	//Delete counters
	IF "DB_ProductionCountersEdit".DeleteCounters > 0 AND "DB_ProductionCountersEdit".DeleteCounters < 4 THEN
	    IF "DB_ProductionCountersEdit".ProgramNumber > 0 AND "DB_ProductionCountersEdit".ProgramNumber <= "NumberOfProductionPrograms" THEN
	        #shiftToDelete := "DB_ProductionCountersEdit".DeleteCounters;
	        "DB_ProductionCountersList".Program["DB_ProductionCountersEdit".ProgramNumber].Product[1].Shift[#shiftToDelete].Ok := 0;
	        "DB_ProductionCountersList".Program["DB_ProductionCountersEdit".ProgramNumber].Product[1].Shift[#shiftToDelete].Nok := 0;
	        "DB_ProductionCountersEdit".ProductCounters := "DB_ProductionCountersList".Program["DB_ProductionCountersEdit".ProgramNumber];
	        FOR #i := 1 TO 50 DO
	            "PartErrorsCounter".CountersRef["DB_ProductionCountersEdit".ProgramNumber].Counters[#shiftToDelete, #i] := 0;
	        END_FOR;
	    END_IF;
	    "DB_ProductionCountersEdit".DeleteCounters := 0;
	END_IF;
	        
	    
	//Auto reset shift counters
	IF "DB_DateTimeAndShifts_Instance".ShiftStatus.Shift1Started THEN
	    FOR #i := 1 TO "NumberOfProductionPrograms" DO
	        "DB_ProductionCountersList".Program[#i].Product[1].Shift[1].Ok := 0;
	        "DB_ProductionCountersList".Program[#i].Product[1].Shift[1].Nok := 0;
	    END_FOR;
	END_IF;
	IF "DB_DateTimeAndShifts_Instance".ShiftStatus.Shift2Started THEN
	    FOR #i := 1 TO "NumberOfProductionPrograms" DO
	        "DB_ProductionCountersList".Program[#i].Product[1].Shift[2].Ok := 0;
	        "DB_ProductionCountersList".Program[#i].Product[1].Shift[2].Nok := 0;
	    END_FOR;
	END_IF;
	IF "DB_DateTimeAndShifts_Instance".ShiftStatus.Shift3Started THEN
	    FOR #i := 1 TO "NumberOfProductionPrograms" DO
	        "DB_ProductionCountersList".Program[#i].Product[1].Shift[3].Ok := 0;
	        "DB_ProductionCountersList".Program[#i].Product[1].Shift[3].Nok := 0;
	    END_FOR;
	END_IF;
	
END_FUNCTION_BLOCK

FUNCTION "PartErrorsCountersMain" : Void
{ S7_Optimized_Access := 'TRUE' }
VERSION : 0.1
   VAR_TEMP 
      i : Int;
   END_VAR


BEGIN
	IF "DB_ProductionCountersEdit".ProgramNumber > 0 AND "DB_ProductionCountersEdit".ProgramNumber <= "NumberOfProductionPrograms" THEN
	    "PartErrorsCounter".CountersHMI := "PartErrorsCounter".CountersRef["DB_ProductionCountersEdit".ProgramNumber];
	END_IF;
	
	
	
	
	
	
	
END_FUNCTION

FUNCTION_BLOCK "FB_Devices"   // FB5100, LAD
{ S7_Optimized_Access := 'TRUE' }
VERSION : 0.1
// stored: AutoNumber false, IsIECCheckEnabled false, IsRetainMemResEnabled false, MemoryReserve 100, SetENOAutomatically false, UDAEnableTagReadback false
   VAR
      ServiceDoors_Instance_1 { S7_SetPoint := 'True'} : "serviceDoor";
      ServiceDoors_Instance_2 { S7_SetPoint := 'True'} : "serviceDoor";
      R_TRIG_Instance { S7_SetPoint := 'True'} : R_TRIG;
      HydraulicActive { S7_SetPoint := 'True'} : Bool;
      HydraulicActiveOffMem : Bool;
      HydraulicOnMem : Bool;
      IEC_Timer_0_Instance { S7_SetPoint := 'True'} : TON_TIME;
      IEC_Timer_0_Instance_1 { S7_SetPoint := 'True'} : TON_TIME;
      FB_TurnTable_Instance { S7_SetPoint := 'True'} : "FB_TurnTable";
      F_TRIG_Instance { S7_SetPoint := 'True'} : F_TRIG;
      edges { S7_SetPoint := 'True'} : Array[1..6] of Bool;
      ManualCommandOld : Int;
      R_TRIG_Instance_1 { S7_SetPoint := 'True'} : R_TRIG;
      R_TRIG_Instance_2 { S7_SetPoint := 'True'} : R_TRIG;
      R_TRIG_Instance_3 { S7_SetPoint := 'True'} : R_TRIG;
      R_TRIG_Instance_4 { S7_SetPoint := 'True'} : R_TRIG;
      R_TRIG_Instance_6 { S7_SetPoint := 'True'} : R_TRIG;
      R_TRIG_Instance_7 { S7_SetPoint := 'True'} : R_TRIG;
      R_TRIG_Instance_8 { S7_SetPoint := 'True'} : R_TRIG;
      R_TRIG_Instance_5 { S7_SetPoint := 'True'} : R_TRIG;
      edgesFitting : Array[1..4] of Bool;
      R_TRIG_V240Wp { S7_SetPoint := 'True'} : R_TRIG;
      R_TRIG_V240Bp { S7_SetPoint := 'True'} : R_TRIG;
      ReaderKeyence_Instance { S7_SetPoint := 'True'} : "ReaderKeyence";
      IEC_Timer_0_Instance_2 { S7_SetPoint := 'True'} : TON_TIME;
      FriedrichUnit1_Instance { S7_SetPoint := 'True'} : "FriedrichUnit";
      FriedrichUnit2_Instance { S7_SetPoint := 'True'} : "FriedrichUnit";
      Trig1 { S7_SetPoint := 'True'} : R_TRIG;
      Trig2 { S7_SetPoint := 'True'} : R_TRIG;
      Trig3 { S7_SetPoint := 'True'} : R_TRIG;
      Trig4 { S7_SetPoint := 'True'} : R_TRIG;
      Camera_CAM1 { S7_SetPoint := 'True'} : "Camera";
      Camera_CAM2 { S7_SetPoint := 'True'} : "Camera";
      Camera_CAM3 { S7_SetPoint := 'True'} : "Camera";
      Camera_CAM4 { S7_SetPoint := 'True'} : "Camera";
      RivetingCycleLeft_Instance { S7_SetPoint := 'True'} : "RivetingCycle";
      RivetingCycleRight_Instance { S7_SetPoint := 'True'} : "RivetingCycle";
   END_VAR
   VAR_TEMP
      posTemp : "UDT_PositionData";
      i : Int;
   END_VAR
   VAR_TEMP   // added for the SCL form of the ladder/FBD networks
      _w1 : Bool;
      _w2 : Bool;
      _w3 : Bool;
   END_VAR
BEGIN

REGION Network 1: Diagnostic fieldbus devices
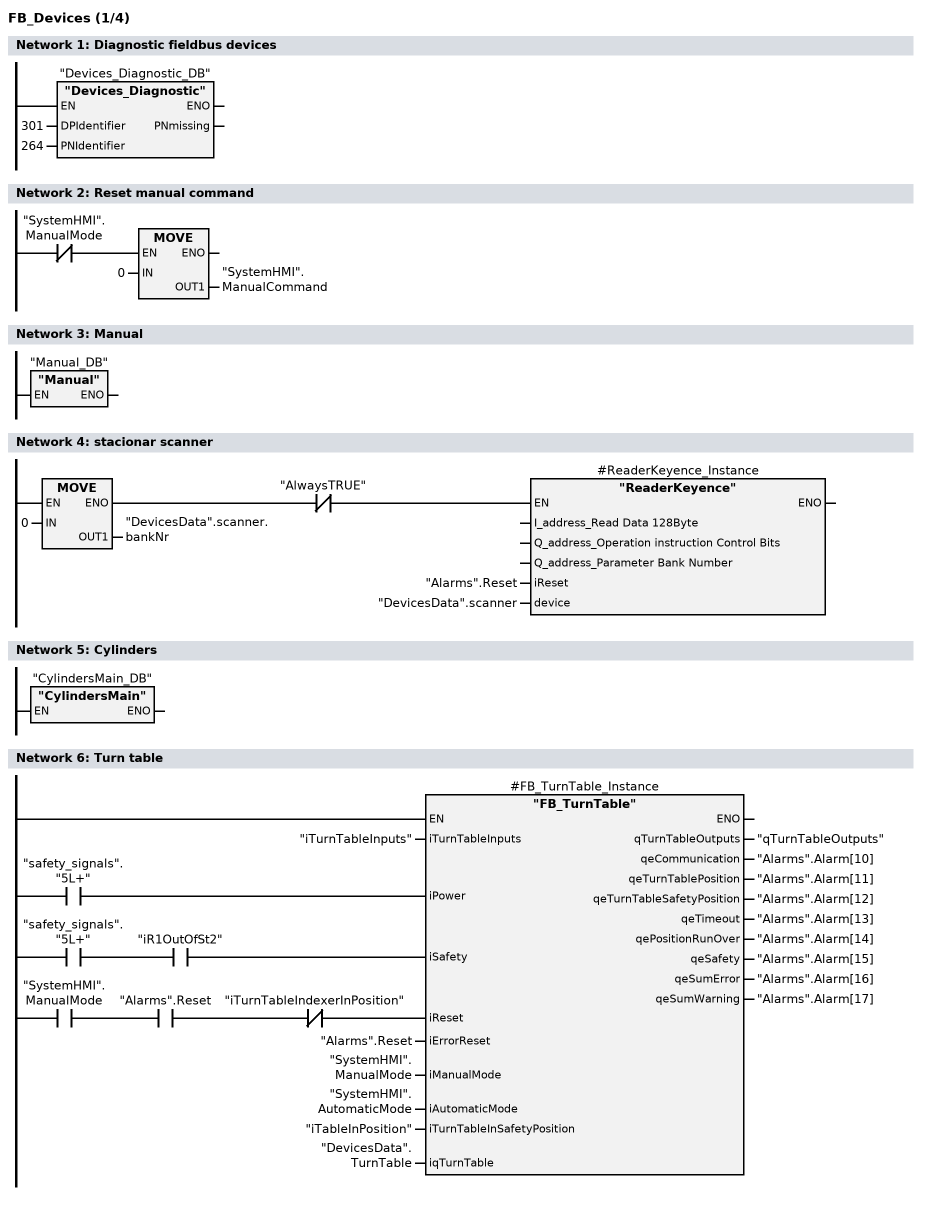
   RUNG wire#powerrail
      "Devices_Diagnostic_DB"(DPIdentifier := 301, PNIdentifier := 264, PNmissing =>)
   END_RUNG
   // the same network as SCL:
   "Devices_Diagnostic_DB"(DPIdentifier := 301, PNIdentifier := 264);   // "Devices_Diagnostic"
END_REGION

REGION Network 2: Reset manual command
   RUNG wire#powerrail
      I_Contact( "SystemHMI".ManualMode )
      Move(in := 0, out1 => "SystemHMI".ManualCommand)
   END_RUNG
   // the same network as SCL:
   IF NOT "SystemHMI".ManualMode THEN "SystemHMI".ManualCommand := 0; END_IF;
END_REGION

REGION Network 3: Manual
   RUNG wire#powerrail
      "Manual_DB"()
   END_RUNG
   // the same network as SCL:
   "Manual_DB"();   // "Manual"
END_REGION

REGION Network 4: stacionar scanner
   RUNG wire#powerrail
      Move(in := 0, out1 => "DevicesData".scanner.bankNr)
      I_Contact( "AlwaysTRUE" )
      #ReaderKeyence_Instance("I_address_Read Data 128Byte" :=, "Q_address_Operation instruction Control Bits" :=, "Q_address_Parameter Bank Number" :=, iReset := "Alarms".Reset, device := "DevicesData".scanner)
   END_RUNG
   // the same network as SCL:
   "DevicesData".scanner.bankNr := 0;
   IF NOT "AlwaysTRUE" THEN
       #ReaderKeyence_Instance(iReset := "Alarms".Reset, device := "DevicesData".scanner);   // "ReaderKeyence"
   END_IF;
END_REGION

REGION Network 5: Cylinders
   RUNG wire#powerrail
      "CylindersMain_DB"()
   END_RUNG
   // the same network as SCL:
   "CylindersMain_DB"();   // "CylindersMain"
END_REGION

REGION Network 6: Turn table
   RUNG wire#powerrail
      #FB_TurnTable_Instance(iPower := wire#w1, iSafety := wire#w2, iReset := wire#w3, iTurnTableInputs := "iTurnTableInputs", iErrorReset := "Alarms".Reset, iManualMode := "SystemHMI".ManualMode, iAutomaticMode := "SystemHMI".AutomaticMode, iTurnTableInSafetyPosition := "iTableInPosition", iqTurnTable := "DevicesData".TurnTable, qTurnTableOutputs => "qTurnTableOutputs", qeCommunication => "Alarms".Alarm[10], qeTurnTablePosition => "Alarms".Alarm[11], qeTurnTableSafetyPosition => "Alarms".Alarm[12], qeTimeout => "Alarms".Alarm[13], qePositionRunOver => "Alarms".Alarm[14], qeSafety => "Alarms".Alarm[15], qeSumError => "Alarms".Alarm[16], qeSumWarning => "Alarms".Alarm[17])
   END_RUNG
   RUNG wire#powerrail
      Contact( "safety_signals"."5L+" )
   END_RUNG wire#w1
   RUNG wire#powerrail
      Contact( "safety_signals"."5L+" )
      Contact( "iR1OutOfSt2" )
   END_RUNG wire#w2
   RUNG wire#powerrail
      Contact( "SystemHMI".ManualMode )
      Contact( "Alarms".Reset )
      I_Contact( "iTurnTableIndexerInPosition" )
   END_RUNG wire#w3
   // the same network as SCL:
   #FB_TurnTable_Instance(iTurnTableInputs := "iTurnTableInputs",   // "FB_TurnTable"
                          iPower := "safety_signals"."5L+",
                          iSafety := "safety_signals"."5L+" AND "iR1OutOfSt2",
                          iReset := "SystemHMI".ManualMode AND "Alarms".Reset AND NOT "iTurnTableIndexerInPosition",
                          iErrorReset := "Alarms".Reset,
                          iManualMode := "SystemHMI".ManualMode,
                          iAutomaticMode := "SystemHMI".AutomaticMode,
                          iTurnTableInSafetyPosition := "iTableInPosition",
                          iqTurnTable := "DevicesData".TurnTable,
                          qTurnTableOutputs => "qTurnTableOutputs",
                          qeCommunication => "Alarms".Alarm[10],
                          qeTurnTablePosition => "Alarms".Alarm[11],
                          qeTurnTableSafetyPosition => "Alarms".Alarm[12],
                          qeTimeout => "Alarms".Alarm[13],
                          qePositionRunOver => "Alarms".Alarm[14],
                          qeSafety => "Alarms".Alarm[15],
                          qeSumError => "Alarms".Alarm[16],
                          qeSumWarning => "Alarms".Alarm[17]);
END_REGION

REGION Network 7: Handle table positions
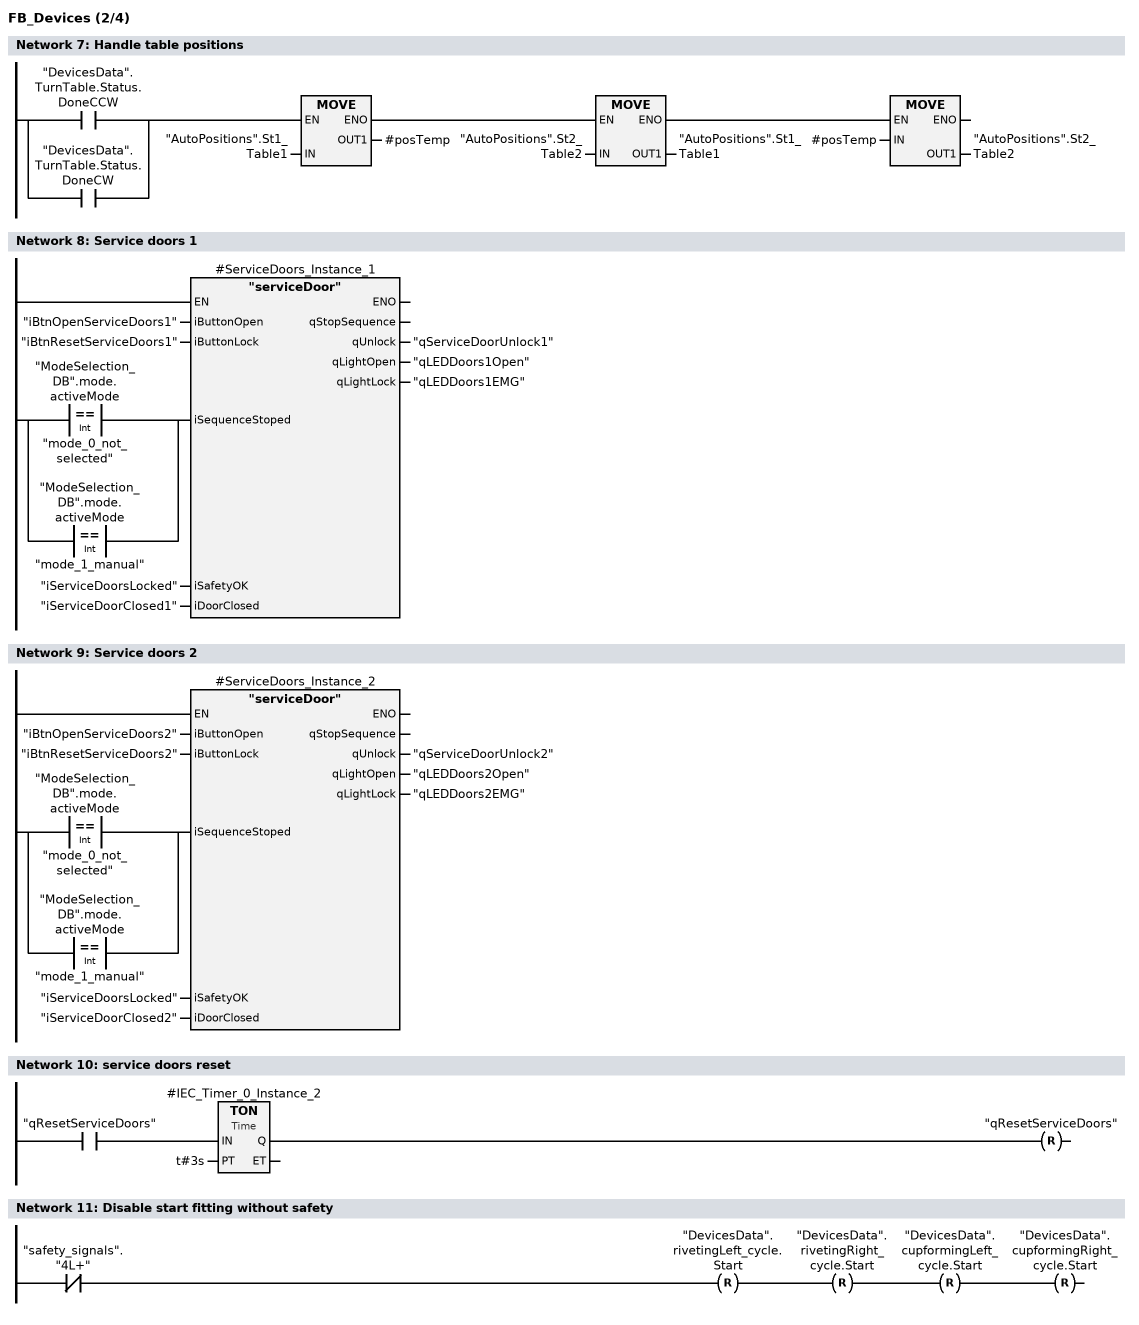
   RUNG wire#powerrail
      Contact( "DevicesData".TurnTable.Status.DoneCCW )
      wire#w1
      Move(in := "AutoPositions".St1_Table1, out1 => #posTemp)
      Move(in := "AutoPositions".St2_Table2, out1 => "AutoPositions".St1_Table1)
      Move(in := #posTemp, out1 => "AutoPositions".St2_Table2)
   END_RUNG
   RUNG wire#powerrail
      Contact( "DevicesData".TurnTable.Status.DoneCW )
   END_RUNG wire#w1
   // the same network as SCL:
   IF "DevicesData".TurnTable.Status.DoneCCW OR "DevicesData".TurnTable.Status.DoneCW THEN
       #posTemp := "AutoPositions".St1_Table1;
       "AutoPositions".St1_Table1 := "AutoPositions".St2_Table2;
       "AutoPositions".St2_Table2 := #posTemp;
   END_IF;
END_REGION

REGION Network 8: Service doors 1
   RUNG wire#powerrail
      #ServiceDoors_Instance_1(iSequenceStoped := wire#w1, iButtonOpen := "iBtnOpenServiceDoors1", iButtonLock := "iBtnResetServiceDoors1", iSafetyOK := "iServiceDoorsLocked", iDoorClosed := "iServiceDoorClosed1", qStopSequence =>, qUnlock => "qServiceDoorUnlock1", qLightOpen => "qLEDDoors1Open", qLightLock => "qLEDDoors1EMG")
   END_RUNG
   RUNG wire#powerrail
      { S7_Templates := "SrcType := Int" } EQ_Contact(in1 := "ModeSelection_DB".mode.activeMode, in2 := "mode_0_not_selected")
   END_RUNG wire#w1
   RUNG wire#powerrail
      { S7_Templates := "SrcType := Int" } EQ_Contact(in1 := "ModeSelection_DB".mode.activeMode, in2 := "mode_1_manual")
   END_RUNG wire#w1
   // the same network as SCL:
   #ServiceDoors_Instance_1(iButtonOpen := "iBtnOpenServiceDoors1",   // "serviceDoor"
                           iButtonLock := "iBtnResetServiceDoors1",
                           iSequenceStoped := ("ModeSelection_DB".mode.activeMode = "mode_0_not_selected") OR ("ModeSelection_DB".mode.activeMode = "mode_1_manual"),
                           iSafetyOK := "iServiceDoorsLocked",
                           iDoorClosed := "iServiceDoorClosed1",
                           qUnlock => "qServiceDoorUnlock1",
                           qLightOpen => "qLEDDoors1Open",
                           qLightLock => "qLEDDoors1EMG");
END_REGION

REGION Network 9: Service doors 2
   RUNG wire#powerrail
      #ServiceDoors_Instance_2(iSequenceStoped := wire#w1, iButtonOpen := "iBtnOpenServiceDoors2", iButtonLock := "iBtnResetServiceDoors2", iSafetyOK := "iServiceDoorsLocked", iDoorClosed := "iServiceDoorClosed2", qStopSequence =>, qUnlock => "qServiceDoorUnlock2", qLightOpen => "qLEDDoors2Open", qLightLock => "qLEDDoors2EMG")
   END_RUNG
   RUNG wire#powerrail
      { S7_Templates := "SrcType := Int" } EQ_Contact(in1 := "ModeSelection_DB".mode.activeMode, in2 := "mode_0_not_selected")
   END_RUNG wire#w1
   RUNG wire#powerrail
      { S7_Templates := "SrcType := Int" } EQ_Contact(in1 := "ModeSelection_DB".mode.activeMode, in2 := "mode_1_manual")
   END_RUNG wire#w1
   // the same network as SCL:
   #ServiceDoors_Instance_2(iButtonOpen := "iBtnOpenServiceDoors2",   // "serviceDoor"
                           iButtonLock := "iBtnResetServiceDoors2",
                           iSequenceStoped := ("ModeSelection_DB".mode.activeMode = "mode_0_not_selected") OR ("ModeSelection_DB".mode.activeMode = "mode_1_manual"),
                           iSafetyOK := "iServiceDoorsLocked",
                           iDoorClosed := "iServiceDoorClosed2",
                           qUnlock => "qServiceDoorUnlock2",
                           qLightOpen => "qLEDDoors2Open",
                           qLightLock => "qLEDDoors2EMG");
END_REGION

REGION Network 10: service doors reset
   RUNG wire#powerrail
      Contact( "qResetServiceDoors" )
      { S7_Templates := "time_type := Time" } #IEC_Timer_0_Instance_2.TON(pt := t#3s, et =>)
      R_Coil( "qResetServiceDoors" )
   END_RUNG
   // the same network as SCL:
   #IEC_Timer_0_Instance_2(IN := "qResetServiceDoors", PT := t#3s);   // TON
   IF #IEC_Timer_0_Instance_2.Q THEN "qResetServiceDoors" := FALSE; END_IF;
END_REGION

REGION Network 11: Disable start fitting without safety
   RUNG wire#powerrail
      I_Contact( "safety_signals"."4L+" )
      R_Coil( "DevicesData".rivetingLeft_cycle.Start )
      R_Coil( "DevicesData".rivetingRight_cycle.Start )
      R_Coil( "DevicesData".cupformingLeft_cycle.Start )
      R_Coil( "DevicesData".cupformingRight_cycle.Start )
   END_RUNG
   // the same network as SCL:
   IF NOT "safety_signals"."4L+" THEN
       "DevicesData".rivetingLeft_cycle.Start := FALSE;
       "DevicesData".rivetingRight_cycle.Start := FALSE;
       "DevicesData".cupformingLeft_cycle.Start := FALSE;
       "DevicesData".cupformingRight_cycle.Start := FALSE;
   END_IF;
END_REGION

REGION Network 12: Fittings - Cyle times measurement
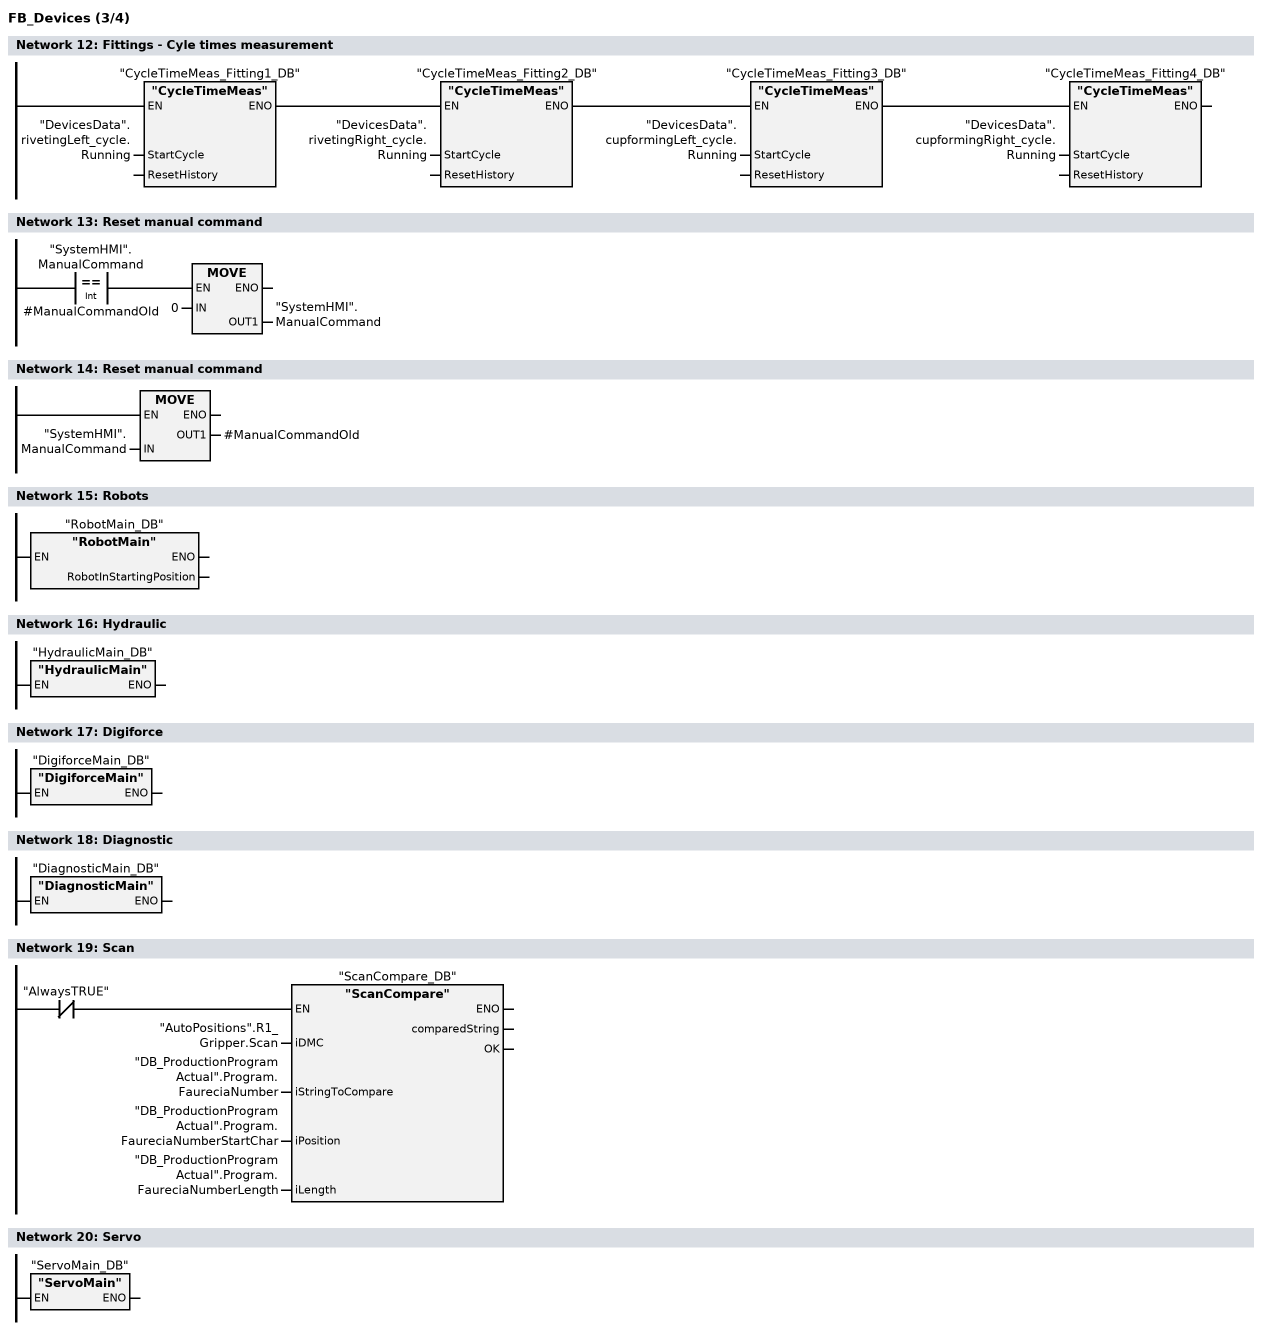
   RUNG wire#powerrail
      "CycleTimeMeas_Fitting1_DB"(StartCycle := "DevicesData".rivetingLeft_cycle.Running, ResetHistory :=)
      "CycleTimeMeas_Fitting2_DB"(StartCycle := "DevicesData".rivetingRight_cycle.Running, ResetHistory :=)
      "CycleTimeMeas_Fitting3_DB"(StartCycle := "DevicesData".cupformingLeft_cycle.Running, ResetHistory :=)
      "CycleTimeMeas_Fitting4_DB"(StartCycle := "DevicesData".cupformingRight_cycle.Running, ResetHistory :=)
   END_RUNG
   // the same network as SCL:
   "CycleTimeMeas_Fitting1_DB"(StartCycle := "DevicesData".rivetingLeft_cycle.Running, ENO => #_w1);   // "CycleTimeMeas"
   "CycleTimeMeas_Fitting2_DB"(EN := #_w1, StartCycle := "DevicesData".rivetingRight_cycle.Running, ENO => #_w2);   // "CycleTimeMeas"
   "CycleTimeMeas_Fitting3_DB"(EN := #_w2,   // "CycleTimeMeas"
                           StartCycle := "DevicesData".cupformingLeft_cycle.Running,
                           ENO => #_w3);
   IF #_w3 THEN
       "CycleTimeMeas_Fitting4_DB"(StartCycle := "DevicesData".cupformingRight_cycle.Running);   // "CycleTimeMeas"
   END_IF;
END_REGION

REGION Network 13: Reset manual command
   RUNG wire#powerrail
      { S7_Templates := "SrcType := Int" } EQ_Contact(in1 := "SystemHMI".ManualCommand, in2 := #ManualCommandOld)
      Move(in := 0, out1 => "SystemHMI".ManualCommand)
   END_RUNG
   // the same network as SCL:
   IF "SystemHMI".ManualCommand = #ManualCommandOld THEN "SystemHMI".ManualCommand := 0; END_IF;
END_REGION

REGION Network 14: Reset manual command
   RUNG wire#powerrail
      Move(in := "SystemHMI".ManualCommand, out1 => #ManualCommandOld)
   END_RUNG
   // the same network as SCL:
   #ManualCommandOld := "SystemHMI".ManualCommand;
END_REGION

REGION Network 15: Robots
   RUNG wire#powerrail
      "RobotMain_DB"(RobotInStartingPosition =>)
   END_RUNG
   // the same network as SCL:
   "RobotMain_DB"();   // "RobotMain"
END_REGION

REGION Network 16: Hydraulic
   RUNG wire#powerrail
      "HydraulicMain_DB"()
   END_RUNG
   // the same network as SCL:
   "HydraulicMain_DB"();   // "HydraulicMain"
END_REGION

REGION Network 17: Digiforce
   RUNG wire#powerrail
      "DigiforceMain_DB"()
   END_RUNG
   // the same network as SCL:
   "DigiforceMain_DB"();   // "DigiforceMain"
END_REGION

REGION Network 18: Diagnostic
   RUNG wire#powerrail
      "DiagnosticMain_DB"()
   END_RUNG
   // the same network as SCL:
   "DiagnosticMain_DB"();   // "DiagnosticMain"
END_REGION

REGION Network 19: Scan
   RUNG wire#powerrail
      I_Contact( "AlwaysTRUE" )
      "ScanCompare_DB"(iDMC := "AutoPositions".R1_Gripper.Scan, iStringToCompare := "DB_ProductionProgramActual".Program.FaureciaNumber, iPosition := "DB_ProductionProgramActual".Program.FaureciaNumberStartChar, iLength := "DB_ProductionProgramActual".Program.FaureciaNumberLength, comparedString =>, OK =>)
   END_RUNG
   // the same network as SCL:
   IF NOT "AlwaysTRUE" THEN
       "ScanCompare_DB"(iDMC := "AutoPositions".R1_Gripper.Scan,   // "ScanCompare"
                        iStringToCompare := "DB_ProductionProgramActual".Program.FaureciaNumber,
                        iPosition := "DB_ProductionProgramActual".Program.FaureciaNumberStartChar,
                        iLength := "DB_ProductionProgramActual".Program.FaureciaNumberLength);
   END_IF;
END_REGION

REGION Network 20: Servo
   RUNG wire#powerrail
      "ServoMain_DB"()
   END_RUNG
   // the same network as SCL:
   "ServoMain_DB"();   // "ServoMain"
END_REGION

REGION Network 21 (SCL): Friedrich1 R
   IF "HMIData".ManualCommand = 611 THEN
       "DevicesData".Friedrich1.Start := true;
   END_IF;

   #FriedrichUnit1_Instance(safetyOK := "safety_signals"."4L+",
                            iReady := "iRivetingReady1",
                            iZ1OK := "iRivetingZ1ok1",
                            iH1OK := "iRivetingH1ok1",
                            iH2OK := "iRivetingH2ok1",
                            iTimeOK := "iRivetingTimeOk1",
                            iNoAlarm := "iRivetingNoError1",
                            FriedrichNumber := 1,
                            Port := 39000,
                            IP1 := 192,
                            IP2 := 168,
                            IP3 := 16,
                            IP4 := 43,
                            ID := 2,
                            qStart => "qRiveting1Start",
                            qPrgbit4 => "qRiveting1Bit4",
                            qPrgbit3 => "qRiveting1Bit3",
                            qPrgbit2 => "qRiveting1Bit2",
                            qPrgbit1 => "qRiveting1Bit1",
                            qPrgbit0 => "qRiveting1Bit0",
                            RivetData := "DevicesData".Friedrich1);
   "qFriedrich1_setup_mode" := "DB_MainData".MachineMode <> 2 AND "DB_MainData".MachineMode <> 3;

   #Trig1(CLK:="DevicesData".Friedrich1.OK);
   #Trig2(CLK:="DevicesData".Friedrich1.NOK);
   "RivetingHistoryRight_DB"(iNewCycle := #Trig1.Q OR #Trig2.Q,
                             iData := "DevicesData".Friedrich1);

   #RivetingCycleRight_Instance(parameters := "DB_ProductionProgramActual".Program.Riveting_program_right,
                                basicPosition := "DevicesData".Friedrich1.Ready AND "DevicesData".Cylinders[MM340_RivetingUnitRight].InBp AND "DevicesData".Cylinders[MM344_RivetingSupportRight].InBp,
                                twoRivets := "DB_ProductionProgramActual".Program.Total_number_of_rivets_4,
                                MeasuredData1=>"AutoInfo".PartMeasuredData.RightRiveting1,
                                MeasuredData2=>"AutoInfo".PartMeasuredData.RightRiveting2,
                                riveter := "DevicesData".Friedrich1,
                                data := "DevicesData".rivetingRight_cycle,
                                cylinderSupport := "DevicesData".Cylinders[MM344_RivetingSupportRight],
                                cylinderShift := "DevicesData".Cylinders[MM340_RivetingUnitRight]);
END_REGION

REGION Network 22 (SCL): Friedrich2 L
   IF "HMIData".ManualCommand = 612 THEN
       "DevicesData".Friedrich2.Start := true;
   END_IF;
   #FriedrichUnit2_Instance(safetyOK := "safety_signals"."4L+",
                            iReady := "iRivetingReady2",
                            iZ1OK := "iRivetingZ1ok2",
                            iH1OK := "iRivetingH1ok2",
                            iH2OK := "iRivetingH2ok2",
                            iTimeOK := "iRivetingTimeOk2",
                            iNoAlarm := "iRivetingNoError2",
                            FriedrichNumber := 2,
                            Port := 39000,
                            IP1 := 192,
                            IP2 := 168,
                            IP3 := 16,
                            IP4 := 44,
                            ID := 3,
                            qStart => "qRiveting2Start",
                            qPrgbit4 => "qRiveting2Bit4",
                            qPrgbit3 => "qRiveting2Bit3",
                            qPrgbit2 => "qRiveting2Bit2",
                            qPrgbit1 => "qRiveting2Bit1",
                            qPrgbit0 => "qRiveting2Bit0",
                            RivetData := "DevicesData".Friedrich2);
   "qFriedrich2_setup_mode" := "DB_MainData".MachineMode <> 2 AND "DB_MainData".MachineMode <> 3;

   #Trig3(CLK:="DevicesData".Friedrich2.OK);
   #Trig4(CLK:="DevicesData".Friedrich2.NOK);
   "RivetingHistoryLeft_DB"(iNewCycle := #Trig3.Q OR #Trig4.Q,
                            iData := "DevicesData".Friedrich2);

   #RivetingCycleLeft_Instance(parameters := "DB_ProductionProgramActual".Program.Riveting_program_left,
                               basicPosition := "DevicesData".Friedrich2.Ready AND "DevicesData".Cylinders[MM342_RivetingUnitLeft].InBp AND "DevicesData".Cylinders[MM346_RivetingSupportLeft].InBp,
                               twoRivets := "DB_ProductionProgramActual".Program.Total_number_of_rivets_4,
                               MeasuredData1=>"AutoInfo".PartMeasuredData.LeftRiveting1,
                               MeasuredData2=>"AutoInfo".PartMeasuredData.LeftRiveting2,
                               riveter := "DevicesData".Friedrich2,
                               data := "DevicesData".rivetingLeft_cycle,
                               cylinderSupport := "DevicesData".Cylinders[MM346_RivetingSupportLeft],
                               cylinderShift := "DevicesData".Cylinders[MM342_RivetingUnitLeft]);

   REGION cycles handshake
       IF "SystemHMI".AutomaticMode THEN
           IF "DevicesData".cupformingLeft_cycle.Done AND "DevicesData".cupformingRight_cycle.Done THEN
               "DevicesData".rivetingLeft_cycle.ContinueFitting := TRUE;
               "DevicesData".rivetingRight_cycle.ContinueFitting := TRUE;
           END_IF;
       END_IF;
       "DevicesData".rivetingLeft_cycle.ContinueFitting := TRUE;
       "DevicesData".rivetingRight_cycle.ContinueFitting := TRUE;

       IF "SystemHMI".ManualMode THEN
           "DevicesData".rivetingLeft_cycle.ContinueFitting := true;
           "DevicesData".rivetingRight_cycle.ContinueFitting := true;
       END_IF;
   END_REGION
END_REGION

REGION Network 23
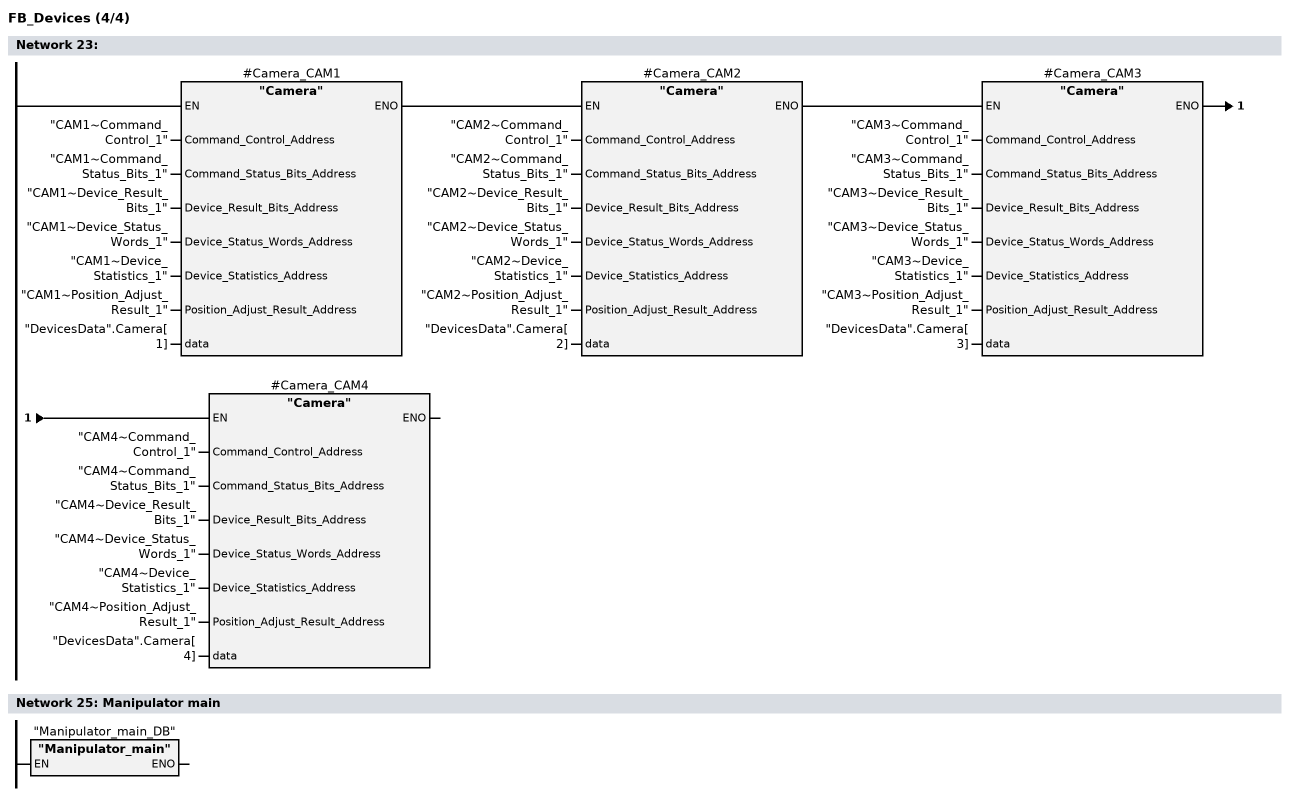
   RUNG wire#powerrail
      #Camera_CAM1(Command_Control_Address := "CAM1~Command_Control_1", Command_Status_Bits_Address := "CAM1~Command_Status_Bits_1", Device_Result_Bits_Address := "CAM1~Device_Result_Bits_1", Device_Status_Words_Address := "CAM1~Device_Status_Words_1", Device_Statistics_Address := "CAM1~Device_Statistics_1", Position_Adjust_Result_Address := "CAM1~Position_Adjust_Result_1", data := "DevicesData".Camera[1])
      #Camera_CAM2(Command_Control_Address := "CAM2~Command_Control_1", Command_Status_Bits_Address := "CAM2~Command_Status_Bits_1", Device_Result_Bits_Address := "CAM2~Device_Result_Bits_1", Device_Status_Words_Address := "CAM2~Device_Status_Words_1", Device_Statistics_Address := "CAM2~Device_Statistics_1", Position_Adjust_Result_Address := "CAM2~Position_Adjust_Result_1", data := "DevicesData".Camera[2])
      #Camera_CAM3(Command_Control_Address := "CAM3~Command_Control_1", Command_Status_Bits_Address := "CAM3~Command_Status_Bits_1", Device_Result_Bits_Address := "CAM3~Device_Result_Bits_1", Device_Status_Words_Address := "CAM3~Device_Status_Words_1", Device_Statistics_Address := "CAM3~Device_Statistics_1", Position_Adjust_Result_Address := "CAM3~Position_Adjust_Result_1", data := "DevicesData".Camera[3])
      #Camera_CAM4(Command_Control_Address := "CAM4~Command_Control_1", Command_Status_Bits_Address := "CAM4~Command_Status_Bits_1", Device_Result_Bits_Address := "CAM4~Device_Result_Bits_1", Device_Status_Words_Address := "CAM4~Device_Status_Words_1", Device_Statistics_Address := "CAM4~Device_Statistics_1", Position_Adjust_Result_Address := "CAM4~Position_Adjust_Result_1", data := "DevicesData".Camera[4])
   END_RUNG
   // the same network as SCL:
   #Camera_CAM1(Command_Control_Address := "CAM1~Command_Control_1",   // "Camera"
                Command_Status_Bits_Address := "CAM1~Command_Status_Bits_1",
                Device_Result_Bits_Address := "CAM1~Device_Result_Bits_1",
                Device_Status_Words_Address := "CAM1~Device_Status_Words_1",
                Device_Statistics_Address := "CAM1~Device_Statistics_1",
                Position_Adjust_Result_Address := "CAM1~Position_Adjust_Result_1",
                data := "DevicesData".Camera[1],
                ENO => #_w1);
   #Camera_CAM2(EN := #_w1,   // "Camera"
                Command_Control_Address := "CAM2~Command_Control_1",
                Command_Status_Bits_Address := "CAM2~Command_Status_Bits_1",
                Device_Result_Bits_Address := "CAM2~Device_Result_Bits_1",
                Device_Status_Words_Address := "CAM2~Device_Status_Words_1",
                Device_Statistics_Address := "CAM2~Device_Statistics_1",
                Position_Adjust_Result_Address := "CAM2~Position_Adjust_Result_1",
                data := "DevicesData".Camera[2],
                ENO => #_w2);
   #Camera_CAM3(EN := #_w2,   // "Camera"
                Command_Control_Address := "CAM3~Command_Control_1",
                Command_Status_Bits_Address := "CAM3~Command_Status_Bits_1",
                Device_Result_Bits_Address := "CAM3~Device_Result_Bits_1",
                Device_Status_Words_Address := "CAM3~Device_Status_Words_1",
                Device_Statistics_Address := "CAM3~Device_Statistics_1",
                Position_Adjust_Result_Address := "CAM3~Position_Adjust_Result_1",
                data := "DevicesData".Camera[3],
                ENO => #_w3);
   IF #_w3 THEN
       #Camera_CAM4(Command_Control_Address := "CAM4~Command_Control_1",   // "Camera"
                    Command_Status_Bits_Address := "CAM4~Command_Status_Bits_1",
                    Device_Result_Bits_Address := "CAM4~Device_Result_Bits_1",
                    Device_Status_Words_Address := "CAM4~Device_Status_Words_1",
                    Device_Statistics_Address := "CAM4~Device_Statistics_1",
                    Position_Adjust_Result_Address := "CAM4~Position_Adjust_Result_1",
                    data := "DevicesData".Camera[4]);
   END_IF;
END_REGION

REGION Network 24 (SCL)
   "DevicesData".Camera[1].ProgramNumber := USINT_TO_SINT("DB_ProductionProgramActual".Program.Camera_program[1]);
   "DevicesData".Camera[2].ProgramNumber := USINT_TO_SINT("DB_ProductionProgramActual".Program.Camera_program[2]);
   "DevicesData".Camera[3].ProgramNumber := USINT_TO_SINT("DB_ProductionProgramActual".Program.Camera_program[3]);
   "DevicesData".Camera[4].ProgramNumber := USINT_TO_SINT("DB_ProductionProgramActual".Program.Camera_program[4]);
END_REGION

REGION Network 25: Manipulator main
   RUNG wire#powerrail
      "Manipulator_main_DB"()
   END_RUNG
   // the same network as SCL:
   "Manipulator_main_DB"();   // "Manipulator_main"
END_REGION

REGION Network 26: Readers
END_REGION
END_FUNCTION_BLOCK

FUNCTION_BLOCK "Devices_Diagnostic"
{ S7_Optimized_Access := 'TRUE' }
VERSION : 0.1
   VAR_INPUT 
      DPIdentifier : HW_IOSYSTEM;
      PNIdentifier : HW_IOSYSTEM;
   END_VAR

   VAR_OUTPUT 
      PNmissing : Bool;
   END_VAR

   VAR 
      PNConfigured : Array[0..1023] of Bool;
      PNFaulty : Array[0..1023] of Bool;
      PNDisabled : Array[0..1023] of Bool;
      PNExist : Array[0..1023] of Bool;
      DPConfigured : Array[0..1023] of Bool;
      DPFaulty : Array[0..1023] of Bool;
      DPDisabled : Array[0..1023] of Bool;
      DPExist : Array[0..1023] of Bool;
   END_VAR

   VAR_TEMP 
      ret : Int;
   END_VAR


BEGIN
	IF #PNIdentifier > 0 THEN
	    #ret := DeviceStates(LADDR := #PNIdentifier, MODE := 1, STATE := #PNConfigured);
	    #ret := DeviceStates(LADDR := #PNIdentifier, MODE := 2, STATE := #PNFaulty);
	    #ret := DeviceStates(LADDR := #PNIdentifier, MODE := 3, STATE := #PNDisabled);
	    #ret := DeviceStates(LADDR := #PNIdentifier, MODE := 4, STATE := #PNExist);
	END_IF;
	
	IF #DPIdentifier > 0 THEN
	    #ret := DeviceStates(LADDR := #DPIdentifier, MODE := 1, STATE := #DPConfigured);
	    #ret := DeviceStates(LADDR := #DPIdentifier, MODE := 2, STATE := #DPFaulty);
	    #ret := DeviceStates(LADDR := #DPIdentifier, MODE := 3, STATE := #DPDisabled);
	    #ret := DeviceStates(LADDR := #DPIdentifier, MODE := 4, STATE := #DPExist);
	END_IF;
	
	#PNmissing := #PNConfigured <> #PNExist;
END_FUNCTION_BLOCK

FUNCTION_BLOCK "Manual"
{ S7_Optimized_Access := 'TRUE' }
VERSION : 0.1
   VAR 
      res : Bool;
      R_TRIG_MM220bp {InstructionName := 'R_TRIG'; LibVersion := '1.0'} : R_TRIG;
      R_TRIG_MM220wp {InstructionName := 'R_TRIG'; LibVersion := '1.0'} : R_TRIG;
      R_TRIG_MM222bp {InstructionName := 'R_TRIG'; LibVersion := '1.0'} : R_TRIG;
      R_TRIG_MM222wp {InstructionName := 'R_TRIG'; LibVersion := '1.0'} : R_TRIG;
      R_TRIG_MM224bp {InstructionName := 'R_TRIG'; LibVersion := '1.0'} : R_TRIG;
      R_TRIG_MM224wp {InstructionName := 'R_TRIG'; LibVersion := '1.0'} : R_TRIG;
   END_VAR


BEGIN
	
	REGION hydraulics
	    IF "HMIData".ManualCommand = 10012 THEN
	        "DevicesData".Hydraulic.StartMotor := true;
	    END_IF;
	    IF "HMIData".ManualCommand = 10011 THEN
	        "DevicesData".Hydraulic.StartMotor := FALSE;
	    END_IF;
	    IF "iOilTemperature65" OR NOT "iOilLowLevelOK" OR NOT "iOilHighLevekOK" THEN
	        "DevicesData".Hydraulic.StartMotor := FALSE;
	    END_IF;
	END_REGION
	
	REGION DMC scanner
	    IF "SystemHMI".ManualMode THEN
	        IF "HMIData".ManualCommand = 3015 THEN
	            "DevicesData".scanner.start := TRUE;
	        END_IF;
	        IF "DevicesData".scanner.newData THEN
	            "AutoInfo".ExtractedScan := "DevicesData".scanner.data;
	        END_IF;
	    END_IF;
	END_REGION
	REGION robot
	    IF "ModeSelection_DB".mode.activeMode = "mode_1_manual" OR NOT "ModeSelection_DB".mode.switch.auto  OR
	        "ModeSelection_DB".mode.activeMode = "mode_0_not_selected" THEN
	        #R_TRIG_MM220bp(CLK := "iR1_MM220grippingTubeToBp");
	        #R_TRIG_MM220wp(CLK := "iR1_MM220grippingTubeToWp");
	        #R_TRIG_MM222bp(CLK := "iR1_MM222holdingSidememberInsideToBp");
	        #R_TRIG_MM222wp(CLK := "iR1_MM222holdingSidememberInsideToWp");
	        #R_TRIG_MM224bp(CLK := "iR1_MM224holdingSidememberOutsideToBp");
	        #R_TRIG_MM224wp(CLK := "iR1_MM224holdingSidememberOutsideToWp");
	        IF #R_TRIG_MM220bp.Q THEN
	            "HMIData".ManualCommand := 1000;
	        END_IF;
	        IF #R_TRIG_MM220wp.Q THEN
	            "HMIData".ManualCommand := 2000;
	        END_IF;
	        IF #R_TRIG_MM222bp.Q THEN
	            "HMIData".ManualCommand := 1002;
	        END_IF;
	        IF #R_TRIG_MM222wp.Q THEN
	            "HMIData".ManualCommand := 2002;
	        END_IF;
	        IF #R_TRIG_MM224bp.Q THEN
	            "HMIData".ManualCommand := 1004;
	        END_IF;
	        IF #R_TRIG_MM224wp.Q THEN
	            "HMIData".ManualCommand := 2004;
	        END_IF;
	    END_IF;
	END_REGION
	
END_FUNCTION_BLOCK

FUNCTION_BLOCK "ReaderKeyence"
{ S7_Optimized_Access := 'TRUE' }
VERSION : 0.1
   VAR_INPUT 
      "I_address_Read Data 128Byte" : HW_IO;
      "Q_address_Operation instruction Control Bits" : HW_IO;
      "Q_address_Parameter Bank Number" : HW_IO;
      iReset : Bool;
   END_VAR

   VAR_IN_OUT 
      device : "UDT_Reader";
   END_VAR

   VAR 
      ResultData : Array[1..128] of Char;
      ResultDataReadyCountOld : UInt;
      R_TRIG_Instance {InstructionName := 'R_TRIG'; LibVersion := '1.0'} : R_TRIG;
      IEC_Timer_0_Instance {InstructionName := 'TON_TIME'; LibVersion := '1.0'} : TON_TIME;
   END_VAR

   VAR_TEMP 
      "Read Data 128ByteTemp" : Struct
         SlaveID : UInt;
         ResultDataReadyCount : UInt;
         ResultDataUpdateCount : UInt;
         ResultDataSize : UInt;
         ResultData : Array[1..128] of Char;
      END_STRUCT;
      "Operation instruction Control Bits" : Struct
         "Read Request" : Bool;
      END_STRUCT;
      retvalTmp : Int;
      i : USInt;
   END_VAR


BEGIN
	#retvalTmp := DPRD_DAT(LADDR := #"I_address_Read Data 128Byte", RECORD => #"Read Data 128ByteTemp");
	
	#R_TRIG_Instance(CLK := #device.start);
	
	#"Operation instruction Control Bits"."Read Request" := #device.start;
	
	IF #R_TRIG_Instance.Q THEN
	    FILL_BLK(IN := ' ',
	             COUNT := 128,
	             OUT => #ResultData[1]);
	    #device.data := '';
	    #device.length := 0;
	END_IF;
	
	#device.newData := FALSE;
	IF #device.start AND #ResultDataReadyCountOld <> #"Read Data 128ByteTemp".ResultDataReadyCount THEN
	    #ResultData := #"Read Data 128ByteTemp".ResultData;
	    #device.length := UINT_TO_USINT(#"Read Data 128ByteTemp".ResultDataSize - 1);
	    FOR #i := 1 TO #device.length DO
	        #device.data[#i] := #ResultData[#i];
	    END_FOR;
	    #device.start := FALSE;
	    #device.newData := TRUE;
	END_IF;
	
	#IEC_Timer_0_Instance(IN:=#device.start,
	                      PT:=t#5s);
	
	IF #IEC_Timer_0_Instance.Q THEN
	    #device.start := FALSE;
	    #device.error := TRUE;
	END_IF;
	
	IF #iReset THEN
	    #device.error := FALSE;
	END_IF;
	
	#ResultDataReadyCountOld := #"Read Data 128ByteTemp".ResultDataReadyCount;
	
	#retvalTmp := DPWR_DAT(LADDR := #"Q_address_Parameter Bank Number", RECORD := #device.bankNr);
	#retvalTmp := DPWR_DAT(LADDR := #"Q_address_Operation instruction Control Bits", RECORD := #"Operation instruction Control Bits");
	
	
	
	
END_FUNCTION_BLOCK

FUNCTION_BLOCK "FB_TurnTable"   // FB3600, LAD
{ S7_Optimized_Access := 'TRUE' }
VERSION : 0.1
// stored: AutoNumber false, IsIECCheckEnabled false, IsRetainMemResEnabled false, MemoryReserve 100, SetENOAutomatically false, UDAEnableTagReadback false
   VAR_INPUT
      iTurnTableInputs : Word;
      iPower : Bool;
      iSafety : Bool;
      iReset : Bool;
      iErrorReset : Bool;
      iManualMode : Bool;
      iAutomaticMode : Bool;
      iTurnTableInSafetyPosition : Bool;
   END_VAR
   VAR_OUTPUT
      qTurnTableOutputs : Word;
      qeCommunication : Bool;
      qeTurnTablePosition : Bool;
      qeTurnTableSafetyPosition : Bool;
      qeTimeout : Bool;
      qePositionRunOver : Bool;
      qeSafety : Bool;
      qeSumError : Bool;
      qeSumWarning : Bool;
   END_VAR
   VAR_IN_OUT
      iqTurnTable : "UDT_TurnTable";
   END_VAR
   VAR
      Edges : Struct
         Enabled : Bool;
         IndexerInPosition : Bool;
      END_STRUCT;
      TONs : Struct
         tDelayCommunication : TON_TIME;
         tDelayPositionError { S7_SetPoint := 'True'} : TON_TIME;
         tDelayErrorReset { S7_SetPoint := 'True'} : TON_TIME;
      END_STRUCT;
   END_VAR
   VAR RETAIN
      RetentiveData : Struct
         LastDirection : Bool;
      END_STRUCT;
   END_VAR
   VAR
      Commands : "UDT_TurnTableCommands";
   END_VAR
   VAR_TEMP
      mode_status : Struct
         manual_mode : Bool;
         automatic_mode : Bool;
         mode_active : Bool;
      END_STRUCT;
      bit : Bool;
      error : Bool;
      ready_to_cw : Bool;
      ready_to_ccw : Bool;
      ready_to_jog : Bool;
      ready_to_start : Bool;
   END_VAR
   VAR_TEMP   // added for the SCL form of the ladder/FBD networks
      _w1 : Bool;
      _w2 : Bool;
      _w3 : Bool;
   END_VAR
BEGIN

REGION Network 1: Read inputs
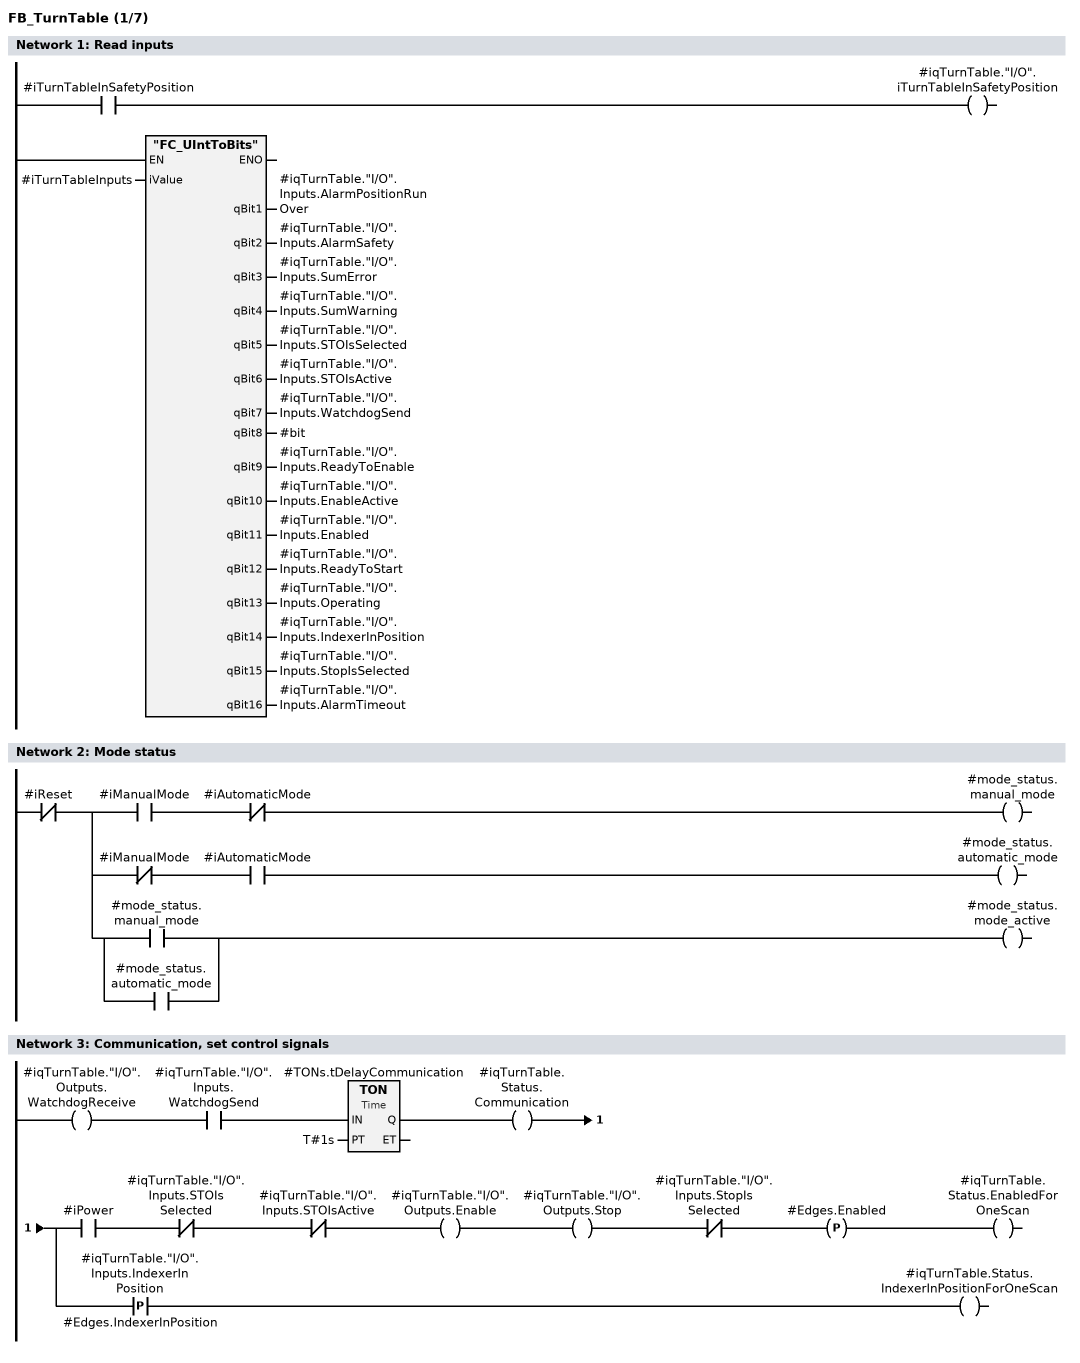
   RUNG wire#powerrail
      Contact( #iTurnTableInSafetyPosition )
      Coil( #iqTurnTable."I/O".iTurnTableInSafetyPosition )
   END_RUNG
   RUNG wire#powerrail
      "FC_UIntToBits"(iValue := #iTurnTableInputs, qBit1 => #iqTurnTable."I/O".Inputs.AlarmPositionRunOver, qBit2 => #iqTurnTable."I/O".Inputs.AlarmSafety, qBit3 => #iqTurnTable."I/O".Inputs.SumError, qBit4 => #iqTurnTable."I/O".Inputs.SumWarning, qBit5 => #iqTurnTable."I/O".Inputs.STOIsSelected, qBit6 => #iqTurnTable."I/O".Inputs.STOIsActive, qBit7 => #iqTurnTable."I/O".Inputs.WatchdogSend, qBit8 => #bit, qBit9 => #iqTurnTable."I/O".Inputs.ReadyToEnable, qBit10 => #iqTurnTable."I/O".Inputs.EnableActive, qBit11 => #iqTurnTable."I/O".Inputs.Enabled, qBit12 => #iqTurnTable."I/O".Inputs.ReadyToStart, qBit13 => #iqTurnTable."I/O".Inputs.Operating, qBit14 => #iqTurnTable."I/O".Inputs.IndexerInPosition, qBit15 => #iqTurnTable."I/O".Inputs.StopIsSelected, qBit16 => #iqTurnTable."I/O".Inputs.AlarmTimeout)
   END_RUNG
   // the same network as SCL:
   #iqTurnTable."I/O".iTurnTableInSafetyPosition := #iTurnTableInSafetyPosition;
   "FC_UIntToBits"(iValue := #iTurnTableInputs,
                   qBit1 => #iqTurnTable."I/O".Inputs.AlarmPositionRunOver,
                   qBit2 => #iqTurnTable."I/O".Inputs.AlarmSafety,
                   qBit3 => #iqTurnTable."I/O".Inputs.SumError,
                   qBit4 => #iqTurnTable."I/O".Inputs.SumWarning,
                   qBit5 => #iqTurnTable."I/O".Inputs.STOIsSelected,
                   qBit6 => #iqTurnTable."I/O".Inputs.STOIsActive,
                   qBit7 => #iqTurnTable."I/O".Inputs.WatchdogSend,
                   qBit8 => #bit,
                   qBit9 => #iqTurnTable."I/O".Inputs.ReadyToEnable,
                   qBit10 => #iqTurnTable."I/O".Inputs.EnableActive,
                   qBit11 => #iqTurnTable."I/O".Inputs.Enabled,
                   qBit12 => #iqTurnTable."I/O".Inputs.ReadyToStart,
                   qBit13 => #iqTurnTable."I/O".Inputs.Operating,
                   qBit14 => #iqTurnTable."I/O".Inputs.IndexerInPosition,
                   qBit15 => #iqTurnTable."I/O".Inputs.StopIsSelected,
                   qBit16 => #iqTurnTable."I/O".Inputs.AlarmTimeout);
END_REGION

REGION Network 2: Mode status
   RUNG wire#powerrail
      I_Contact( #iReset )
      wire#w1
      Contact( #iManualMode )
      I_Contact( #iAutomaticMode )
      Coil( #mode_status.manual_mode )
   END_RUNG
   RUNG wire#w1
      I_Contact( #iManualMode )
      Contact( #iAutomaticMode )
      Coil( #mode_status.automatic_mode )
   END_RUNG
   RUNG wire#w1
      Contact( #mode_status.manual_mode )
      wire#w2
      Coil( #mode_status.mode_active )
   END_RUNG
   RUNG wire#w1
      Contact( #mode_status.automatic_mode )
   END_RUNG wire#w2
   // the same network as SCL:
   #mode_status.manual_mode := NOT #iReset AND #iManualMode AND NOT #iAutomaticMode;
   #mode_status.automatic_mode := NOT #iReset AND NOT #iManualMode AND #iAutomaticMode;
   #mode_status.mode_active := NOT #iReset AND (#mode_status.manual_mode OR #mode_status.automatic_mode);
END_REGION

REGION Network 3: Communication, set control signals
   RUNG wire#powerrail
      Coil( #iqTurnTable."I/O".Outputs.WatchdogReceive )
      Contact( #iqTurnTable."I/O".Inputs.WatchdogSend )
      { S7_Templates := "time_type := Time" } #TONs.tDelayCommunication.TON(pt := T#1s, et =>)
      Coil( #iqTurnTable.Status.Communication )
      wire#w1
      Contact( #iPower )
      I_Contact( #iqTurnTable."I/O".Inputs.STOIsSelected )
      I_Contact( #iqTurnTable."I/O".Inputs.STOIsActive )
      Coil( #iqTurnTable."I/O".Outputs.Enable )
      Coil( #iqTurnTable."I/O".Outputs.Stop )
      I_Contact( #iqTurnTable."I/O".Inputs.StopIsSelected )
      P_Trig( #Edges.Enabled )
      Coil( #iqTurnTable.Status.EnabledForOneScan )
   END_RUNG
   RUNG wire#w1
      P_Contact(operand := #iqTurnTable."I/O".Inputs.IndexerInPosition, bit := #Edges.IndexerInPosition)
      Coil( #iqTurnTable.Status.IndexerInPositionForOneScan )
   END_RUNG
   // the same network as SCL:
   #iqTurnTable."I/O".Outputs.WatchdogReceive := TRUE;
   #TONs.tDelayCommunication.TON(IN := #iqTurnTable."I/O".Inputs.WatchdogSend, PT := T#1s);
   #iqTurnTable.Status.Communication := #TONs.tDelayCommunication.Q;
   #iqTurnTable."I/O".Outputs.Enable := #TONs.tDelayCommunication.Q AND #iPower AND NOT #iqTurnTable."I/O".Inputs.STOIsSelected AND NOT #iqTurnTable."I/O".Inputs.STOIsActive;
   #iqTurnTable."I/O".Outputs.Stop := #iqTurnTable."I/O".Outputs.Enable;
   #_w1 := #iqTurnTable."I/O".Outputs.Enable AND NOT #iqTurnTable."I/O".Inputs.StopIsSelected;
   #_w2 := #_w1 AND NOT #Edges.Enabled;   // rising edge
   #Edges.Enabled := #_w1;
   #iqTurnTable.Status.EnabledForOneScan := #_w2;
   #_w3 := #TONs.tDelayCommunication.Q AND #iqTurnTable."I/O".Inputs.IndexerInPosition AND NOT #Edges.IndexerInPosition;   // rising edge of #iqTurnTable."I/O".Inputs.IndexerInPosition
   #Edges.IndexerInPosition := #iqTurnTable."I/O".Inputs.IndexerInPosition;
   #iqTurnTable.Status.IndexerInPositionForOneScan := #_w3;
END_REGION

REGION Network 4: Errors
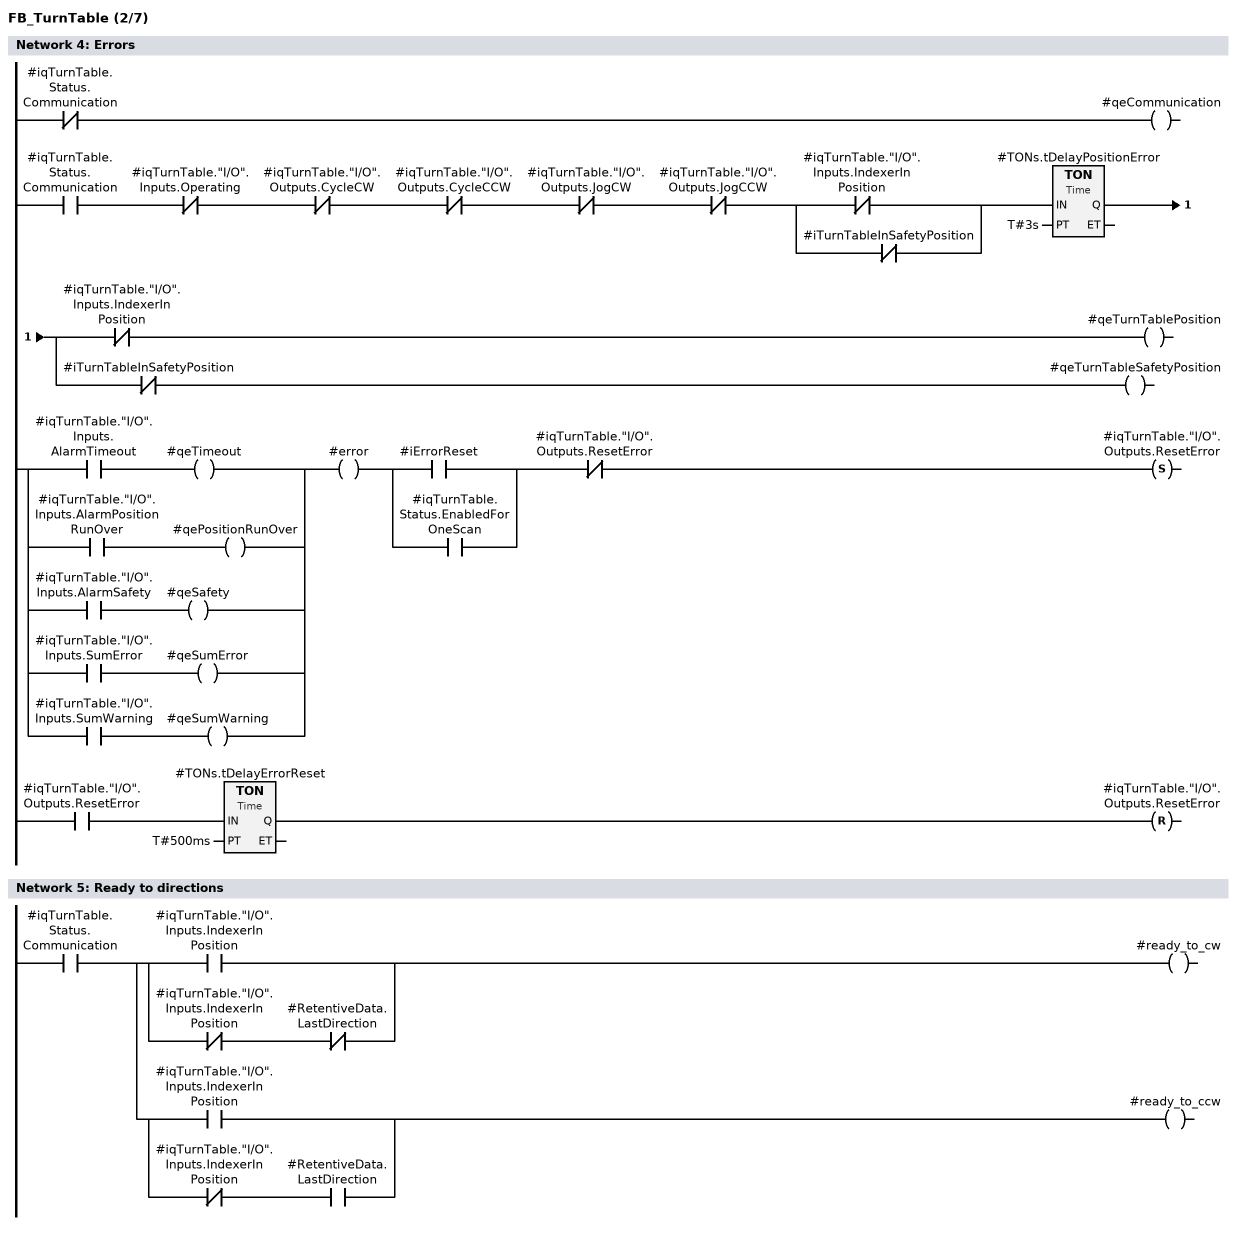
   RUNG wire#powerrail
      I_Contact( #iqTurnTable.Status.Communication )
      Coil( #qeCommunication )
   END_RUNG
   RUNG wire#powerrail
      Contact( #iqTurnTable.Status.Communication )
      I_Contact( #iqTurnTable."I/O".Inputs.Operating )
      I_Contact( #iqTurnTable."I/O".Outputs.CycleCW )
      I_Contact( #iqTurnTable."I/O".Outputs.CycleCCW )
      I_Contact( #iqTurnTable."I/O".Outputs.JogCW )
      I_Contact( #iqTurnTable."I/O".Outputs.JogCCW )
      wire#w1
      I_Contact( #iqTurnTable."I/O".Inputs.IndexerInPosition )
      wire#w2
      { S7_Templates := "time_type := Time" } #TONs.tDelayPositionError.TON(pt := T#3s, et =>)
      wire#w3
      I_Contact( #iqTurnTable."I/O".Inputs.IndexerInPosition )
      Coil( #qeTurnTablePosition )
   END_RUNG
   RUNG wire#w1
      I_Contact( #iTurnTableInSafetyPosition )
   END_RUNG wire#w2
   RUNG wire#w3
      I_Contact( #iTurnTableInSafetyPosition )
      Coil( #qeTurnTableSafetyPosition )
   END_RUNG
   RUNG wire#powerrail
      Contact( #iqTurnTable."I/O".Inputs.AlarmTimeout )
      Coil( #qeTimeout )
      wire#w4
      Coil( #error )
      wire#w5
      Contact( #iErrorReset )
      wire#w6
      I_Contact( #iqTurnTable."I/O".Outputs.ResetError )
      S_Coil( #iqTurnTable."I/O".Outputs.ResetError )
   END_RUNG
   RUNG wire#powerrail
      Contact( #iqTurnTable."I/O".Inputs.AlarmPositionRunOver )
      Coil( #qePositionRunOver )
   END_RUNG wire#w4
   RUNG wire#powerrail
      Contact( #iqTurnTable."I/O".Inputs.AlarmSafety )
      Coil( #qeSafety )
   END_RUNG wire#w4
   RUNG wire#powerrail
      Contact( #iqTurnTable."I/O".Inputs.SumError )
      Coil( #qeSumError )
   END_RUNG wire#w4
   RUNG wire#powerrail
      Contact( #iqTurnTable."I/O".Inputs.SumWarning )
      Coil( #qeSumWarning )
   END_RUNG wire#w4
   RUNG wire#w5
      Contact( #iqTurnTable.Status.EnabledForOneScan )
   END_RUNG wire#w6
   RUNG wire#powerrail
      Contact( #iqTurnTable."I/O".Outputs.ResetError )
      { S7_Templates := "time_type := Time" } #TONs.tDelayErrorReset.TON(pt := T#500ms, et =>)
      R_Coil( #iqTurnTable."I/O".Outputs.ResetError )
   END_RUNG
   // the same network as SCL:
   #qeCommunication := NOT #iqTurnTable.Status.Communication;
   #TONs.tDelayPositionError.TON(IN := #iqTurnTable.Status.Communication AND NOT #iqTurnTable."I/O".Inputs.Operating AND NOT #iqTurnTable."I/O".Outputs.CycleCW AND NOT #iqTurnTable."I/O".Outputs.CycleCCW AND NOT #iqTurnTable."I/O".Outputs.JogCW AND NOT #iqTurnTable."I/O".Outputs.JogCCW AND (NOT #iqTurnTable."I/O".Inputs.IndexerInPosition OR NOT #iTurnTableInSafetyPosition),
                           PT := T#3s);
   #qeTurnTablePosition := #TONs.tDelayPositionError.Q AND NOT #iqTurnTable."I/O".Inputs.IndexerInPosition;
   #qeTurnTableSafetyPosition := #TONs.tDelayPositionError.Q AND NOT #iTurnTableInSafetyPosition;
   #qeTimeout := #iqTurnTable."I/O".Inputs.AlarmTimeout;
   #qePositionRunOver := #iqTurnTable."I/O".Inputs.AlarmPositionRunOver;
   #qeSafety := #iqTurnTable."I/O".Inputs.AlarmSafety;
   #qeSumError := #iqTurnTable."I/O".Inputs.SumError;
   #qeSumWarning := #iqTurnTable."I/O".Inputs.SumWarning;
   #error := #iqTurnTable."I/O".Inputs.AlarmTimeout OR #iqTurnTable."I/O".Inputs.AlarmPositionRunOver OR #iqTurnTable."I/O".Inputs.AlarmSafety OR #iqTurnTable."I/O".Inputs.SumError OR #iqTurnTable."I/O".Inputs.SumWarning;
   IF #error AND (#iErrorReset OR #iqTurnTable.Status.EnabledForOneScan) AND NOT #iqTurnTable."I/O".Outputs.ResetError THEN
       #iqTurnTable."I/O".Outputs.ResetError := TRUE;
   END_IF;
   #TONs.tDelayErrorReset.TON(IN := #iqTurnTable."I/O".Outputs.ResetError, PT := T#500ms);
   IF #TONs.tDelayErrorReset.Q THEN #iqTurnTable."I/O".Outputs.ResetError := FALSE; END_IF;
END_REGION

REGION Network 5: Ready to directions
   RUNG wire#powerrail
      Contact( #iqTurnTable.Status.Communication )
      wire#w1
      Contact( #iqTurnTable."I/O".Inputs.IndexerInPosition )
      wire#w2
      Coil( #ready_to_cw )
   END_RUNG
   RUNG wire#w1
      I_Contact( #iqTurnTable."I/O".Inputs.IndexerInPosition )
      I_Contact( #RetentiveData.LastDirection )
   END_RUNG wire#w2
   RUNG wire#w1
      Contact( #iqTurnTable."I/O".Inputs.IndexerInPosition )
      wire#w3
      Coil( #ready_to_ccw )
   END_RUNG
   RUNG wire#w1
      I_Contact( #iqTurnTable."I/O".Inputs.IndexerInPosition )
      Contact( #RetentiveData.LastDirection )
   END_RUNG wire#w3
   // the same network as SCL:
   #ready_to_cw := #iqTurnTable.Status.Communication AND (#iqTurnTable."I/O".Inputs.IndexerInPosition OR (NOT #iqTurnTable."I/O".Inputs.IndexerInPosition AND NOT #RetentiveData.LastDirection));
   #ready_to_ccw := #iqTurnTable.Status.Communication AND (#iqTurnTable."I/O".Inputs.IndexerInPosition OR (NOT #iqTurnTable."I/O".Inputs.IndexerInPosition AND #RetentiveData.LastDirection));
END_REGION

REGION Network 6: Ready to jog
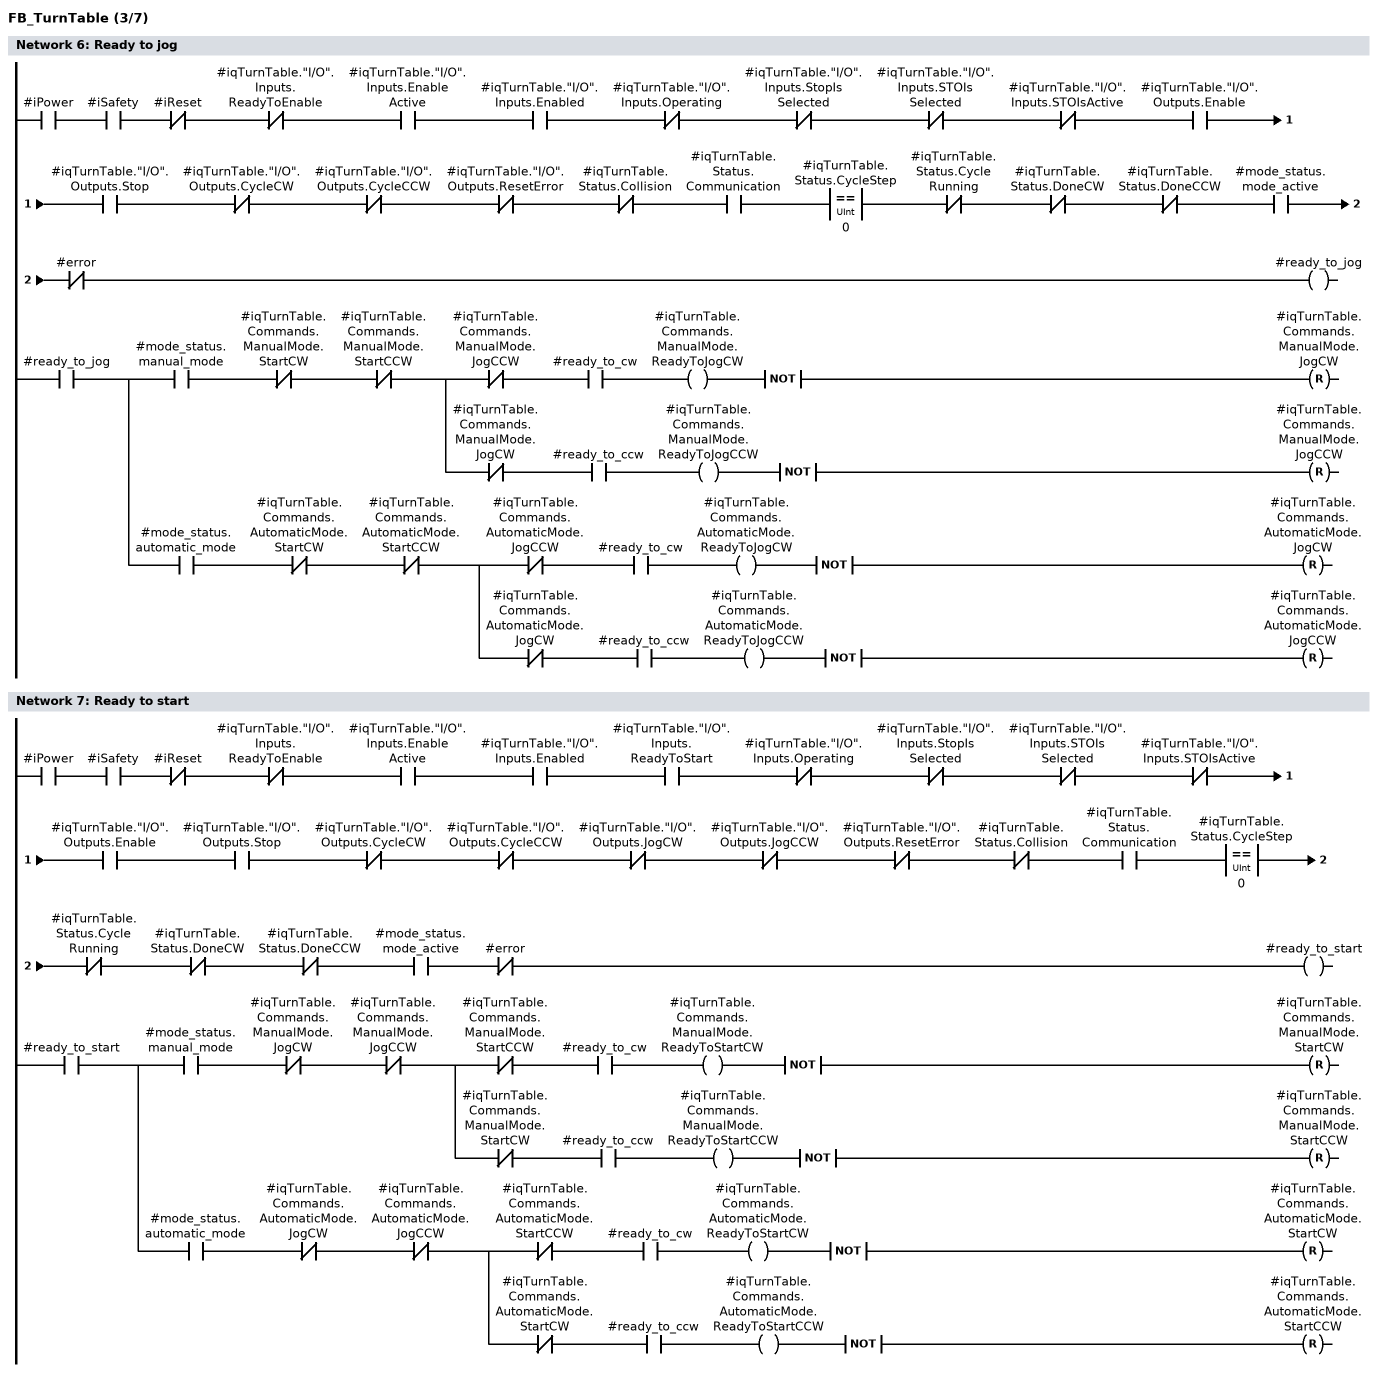
   RUNG wire#powerrail
      Contact( #iPower )
      Contact( #iSafety )
      I_Contact( #iReset )
      I_Contact( #iqTurnTable."I/O".Inputs.ReadyToEnable )
      Contact( #iqTurnTable."I/O".Inputs.EnableActive )
      Contact( #iqTurnTable."I/O".Inputs.Enabled )
      I_Contact( #iqTurnTable."I/O".Inputs.Operating )
      I_Contact( #iqTurnTable."I/O".Inputs.StopIsSelected )
      I_Contact( #iqTurnTable."I/O".Inputs.STOIsSelected )
      I_Contact( #iqTurnTable."I/O".Inputs.STOIsActive )
      Contact( #iqTurnTable."I/O".Outputs.Enable )
      Contact( #iqTurnTable."I/O".Outputs.Stop )
      I_Contact( #iqTurnTable."I/O".Outputs.CycleCW )
      I_Contact( #iqTurnTable."I/O".Outputs.CycleCCW )
      I_Contact( #iqTurnTable."I/O".Outputs.ResetError )
      I_Contact( #iqTurnTable.Status.Collision )
      Contact( #iqTurnTable.Status.Communication )
      { S7_Templates := "SrcType := UInt" } EQ_Contact(in1 := #iqTurnTable.Status.CycleStep, in2 := 0)
      I_Contact( #iqTurnTable.Status.CycleRunning )
      I_Contact( #iqTurnTable.Status.DoneCW )
      I_Contact( #iqTurnTable.Status.DoneCCW )
      Contact( #mode_status.mode_active )
      I_Contact( #error )
      Coil( #ready_to_jog )
   END_RUNG
   RUNG wire#powerrail
      Contact( #ready_to_jog )
      wire#w1
      Contact( #mode_status.manual_mode )
      I_Contact( #iqTurnTable.Commands.ManualMode.StartCW )
      I_Contact( #iqTurnTable.Commands.ManualMode.StartCCW )
      wire#w2
      I_Contact( #iqTurnTable.Commands.ManualMode.JogCCW )
      Contact( #ready_to_cw )
      Coil( #iqTurnTable.Commands.ManualMode.ReadyToJogCW )
      Not()
      R_Coil( #iqTurnTable.Commands.ManualMode.JogCW )
   END_RUNG
   RUNG wire#w2
      I_Contact( #iqTurnTable.Commands.ManualMode.JogCW )
      Contact( #ready_to_ccw )
      Coil( #iqTurnTable.Commands.ManualMode.ReadyToJogCCW )
      Not()
      R_Coil( #iqTurnTable.Commands.ManualMode.JogCCW )
   END_RUNG
   RUNG wire#w1
      Contact( #mode_status.automatic_mode )
      I_Contact( #iqTurnTable.Commands.AutomaticMode.StartCW )
      I_Contact( #iqTurnTable.Commands.AutomaticMode.StartCCW )
      wire#w3
      I_Contact( #iqTurnTable.Commands.AutomaticMode.JogCCW )
      Contact( #ready_to_cw )
      Coil( #iqTurnTable.Commands.AutomaticMode.ReadyToJogCW )
      Not()
      R_Coil( #iqTurnTable.Commands.AutomaticMode.JogCW )
   END_RUNG
   RUNG wire#w3
      I_Contact( #iqTurnTable.Commands.AutomaticMode.JogCW )
      Contact( #ready_to_ccw )
      Coil( #iqTurnTable.Commands.AutomaticMode.ReadyToJogCCW )
      Not()
      R_Coil( #iqTurnTable.Commands.AutomaticMode.JogCCW )
   END_RUNG
   // the same network as SCL:
   #ready_to_jog := #iPower AND #iSafety AND NOT #iReset AND NOT #iqTurnTable."I/O".Inputs.ReadyToEnable AND #iqTurnTable."I/O".Inputs.EnableActive AND #iqTurnTable."I/O".Inputs.Enabled AND NOT #iqTurnTable."I/O".Inputs.Operating AND NOT #iqTurnTable."I/O".Inputs.StopIsSelected AND NOT #iqTurnTable."I/O".Inputs.STOIsSelected AND NOT #iqTurnTable."I/O".Inputs.STOIsActive AND #iqTurnTable."I/O".Outputs.Enable AND #iqTurnTable."I/O".Outputs.Stop AND NOT #iqTurnTable."I/O".Outputs.CycleCW AND NOT #iqTurnTable."I/O".Outputs.CycleCCW AND NOT #iqTurnTable."I/O".Outputs.ResetError AND NOT #iqTurnTable.Status.Collision AND #iqTurnTable.Status.Communication AND (#iqTurnTable.Status.CycleStep = 0) AND NOT #iqTurnTable.Status.CycleRunning AND NOT #iqTurnTable.Status.DoneCW AND NOT #iqTurnTable.Status.DoneCCW AND #mode_status.mode_active AND NOT #error;
   #_w1 := #ready_to_jog AND #mode_status.manual_mode AND NOT #iqTurnTable.Commands.ManualMode.StartCW AND NOT #iqTurnTable.Commands.ManualMode.StartCCW;
   #iqTurnTable.Commands.ManualMode.ReadyToJogCW := #_w1 AND NOT #iqTurnTable.Commands.ManualMode.JogCCW AND #ready_to_cw;
   IF NOT #iqTurnTable.Commands.ManualMode.ReadyToJogCW THEN
       #iqTurnTable.Commands.ManualMode.JogCW := FALSE;
   END_IF;
   #iqTurnTable.Commands.ManualMode.ReadyToJogCCW := #_w1 AND NOT #iqTurnTable.Commands.ManualMode.JogCW AND #ready_to_ccw;
   IF NOT #iqTurnTable.Commands.ManualMode.ReadyToJogCCW THEN
       #iqTurnTable.Commands.ManualMode.JogCCW := FALSE;
   END_IF;
   #_w2 := #ready_to_jog AND #mode_status.automatic_mode AND NOT #iqTurnTable.Commands.AutomaticMode.StartCW AND NOT #iqTurnTable.Commands.AutomaticMode.StartCCW;
   #iqTurnTable.Commands.AutomaticMode.ReadyToJogCW := #_w2 AND NOT #iqTurnTable.Commands.AutomaticMode.JogCCW AND #ready_to_cw;
   IF NOT #iqTurnTable.Commands.AutomaticMode.ReadyToJogCW THEN
       #iqTurnTable.Commands.AutomaticMode.JogCW := FALSE;
   END_IF;
   #iqTurnTable.Commands.AutomaticMode.ReadyToJogCCW := #_w2 AND NOT #iqTurnTable.Commands.AutomaticMode.JogCW AND #ready_to_ccw;
   IF NOT #iqTurnTable.Commands.AutomaticMode.ReadyToJogCCW THEN
       #iqTurnTable.Commands.AutomaticMode.JogCCW := FALSE;
   END_IF;
END_REGION

REGION Network 7: Ready to start
   RUNG wire#powerrail
      Contact( #iPower )
      Contact( #iSafety )
      I_Contact( #iReset )
      I_Contact( #iqTurnTable."I/O".Inputs.ReadyToEnable )
      Contact( #iqTurnTable."I/O".Inputs.EnableActive )
      Contact( #iqTurnTable."I/O".Inputs.Enabled )
      Contact( #iqTurnTable."I/O".Inputs.ReadyToStart )
      I_Contact( #iqTurnTable."I/O".Inputs.Operating )
      I_Contact( #iqTurnTable."I/O".Inputs.StopIsSelected )
      I_Contact( #iqTurnTable."I/O".Inputs.STOIsSelected )
      I_Contact( #iqTurnTable."I/O".Inputs.STOIsActive )
      Contact( #iqTurnTable."I/O".Outputs.Enable )
      Contact( #iqTurnTable."I/O".Outputs.Stop )
      I_Contact( #iqTurnTable."I/O".Outputs.CycleCW )
      I_Contact( #iqTurnTable."I/O".Outputs.CycleCCW )
      I_Contact( #iqTurnTable."I/O".Outputs.JogCW )
      I_Contact( #iqTurnTable."I/O".Outputs.JogCCW )
      I_Contact( #iqTurnTable."I/O".Outputs.ResetError )
      I_Contact( #iqTurnTable.Status.Collision )
      Contact( #iqTurnTable.Status.Communication )
      { S7_Templates := "SrcType := UInt" } EQ_Contact(in1 := #iqTurnTable.Status.CycleStep, in2 := 0)
      I_Contact( #iqTurnTable.Status.CycleRunning )
      I_Contact( #iqTurnTable.Status.DoneCW )
      I_Contact( #iqTurnTable.Status.DoneCCW )
      Contact( #mode_status.mode_active )
      I_Contact( #error )
      Coil( #ready_to_start )
   END_RUNG
   RUNG wire#powerrail
      Contact( #ready_to_start )
      wire#w1
      Contact( #mode_status.manual_mode )
      I_Contact( #iqTurnTable.Commands.ManualMode.JogCW )
      I_Contact( #iqTurnTable.Commands.ManualMode.JogCCW )
      wire#w2
      I_Contact( #iqTurnTable.Commands.ManualMode.StartCCW )
      Contact( #ready_to_cw )
      Coil( #iqTurnTable.Commands.ManualMode.ReadyToStartCW )
      Not()
      R_Coil( #iqTurnTable.Commands.ManualMode.StartCW )
   END_RUNG
   RUNG wire#w2
      I_Contact( #iqTurnTable.Commands.ManualMode.StartCW )
      Contact( #ready_to_ccw )
      Coil( #iqTurnTable.Commands.ManualMode.ReadyToStartCCW )
      Not()
      R_Coil( #iqTurnTable.Commands.ManualMode.StartCCW )
   END_RUNG
   RUNG wire#w1
      Contact( #mode_status.automatic_mode )
      I_Contact( #iqTurnTable.Commands.AutomaticMode.JogCW )
      I_Contact( #iqTurnTable.Commands.AutomaticMode.JogCCW )
      wire#w3
      I_Contact( #iqTurnTable.Commands.AutomaticMode.StartCCW )
      Contact( #ready_to_cw )
      Coil( #iqTurnTable.Commands.AutomaticMode.ReadyToStartCW )
      Not()
      R_Coil( #iqTurnTable.Commands.AutomaticMode.StartCW )
   END_RUNG
   RUNG wire#w3
      I_Contact( #iqTurnTable.Commands.AutomaticMode.StartCW )
      Contact( #ready_to_ccw )
      Coil( #iqTurnTable.Commands.AutomaticMode.ReadyToStartCCW )
      Not()
      R_Coil( #iqTurnTable.Commands.AutomaticMode.StartCCW )
   END_RUNG
   // the same network as SCL:
   #ready_to_start := #iPower AND #iSafety AND NOT #iReset AND NOT #iqTurnTable."I/O".Inputs.ReadyToEnable AND #iqTurnTable."I/O".Inputs.EnableActive AND #iqTurnTable."I/O".Inputs.Enabled AND #iqTurnTable."I/O".Inputs.ReadyToStart AND NOT #iqTurnTable."I/O".Inputs.Operating AND NOT #iqTurnTable."I/O".Inputs.StopIsSelected AND NOT #iqTurnTable."I/O".Inputs.STOIsSelected AND NOT #iqTurnTable."I/O".Inputs.STOIsActive AND #iqTurnTable."I/O".Outputs.Enable AND #iqTurnTable."I/O".Outputs.Stop AND NOT #iqTurnTable."I/O".Outputs.CycleCW AND NOT #iqTurnTable."I/O".Outputs.CycleCCW AND NOT #iqTurnTable."I/O".Outputs.JogCW AND NOT #iqTurnTable."I/O".Outputs.JogCCW AND NOT #iqTurnTable."I/O".Outputs.ResetError AND NOT #iqTurnTable.Status.Collision AND #iqTurnTable.Status.Communication AND (#iqTurnTable.Status.CycleStep = 0) AND NOT #iqTurnTable.Status.CycleRunning AND NOT #iqTurnTable.Status.DoneCW AND NOT #iqTurnTable.Status.DoneCCW AND #mode_status.mode_active AND NOT #error;
   #_w1 := #ready_to_start AND #mode_status.manual_mode AND NOT #iqTurnTable.Commands.ManualMode.JogCW AND NOT #iqTurnTable.Commands.ManualMode.JogCCW;
   #iqTurnTable.Commands.ManualMode.ReadyToStartCW := #_w1 AND NOT #iqTurnTable.Commands.ManualMode.StartCCW AND #ready_to_cw;
   IF NOT #iqTurnTable.Commands.ManualMode.ReadyToStartCW THEN
       #iqTurnTable.Commands.ManualMode.StartCW := FALSE;
   END_IF;
   #iqTurnTable.Commands.ManualMode.ReadyToStartCCW := #_w1 AND NOT #iqTurnTable.Commands.ManualMode.StartCW AND #ready_to_ccw;
   IF NOT #iqTurnTable.Commands.ManualMode.ReadyToStartCCW THEN
       #iqTurnTable.Commands.ManualMode.StartCCW := FALSE;
   END_IF;
   #_w2 := #ready_to_start AND #mode_status.automatic_mode AND NOT #iqTurnTable.Commands.AutomaticMode.JogCW AND NOT #iqTurnTable.Commands.AutomaticMode.JogCCW;
   #iqTurnTable.Commands.AutomaticMode.ReadyToStartCW := #_w2 AND NOT #iqTurnTable.Commands.AutomaticMode.StartCCW AND #ready_to_cw;
   IF NOT #iqTurnTable.Commands.AutomaticMode.ReadyToStartCW THEN
       #iqTurnTable.Commands.AutomaticMode.StartCW := FALSE;
   END_IF;
   #iqTurnTable.Commands.AutomaticMode.ReadyToStartCCW := #_w2 AND NOT #iqTurnTable.Commands.AutomaticMode.StartCW AND #ready_to_ccw;
   IF NOT #iqTurnTable.Commands.AutomaticMode.ReadyToStartCCW THEN
       #iqTurnTable.Commands.AutomaticMode.StartCCW := FALSE;
   END_IF;
END_REGION

REGION Network 8: Set commands
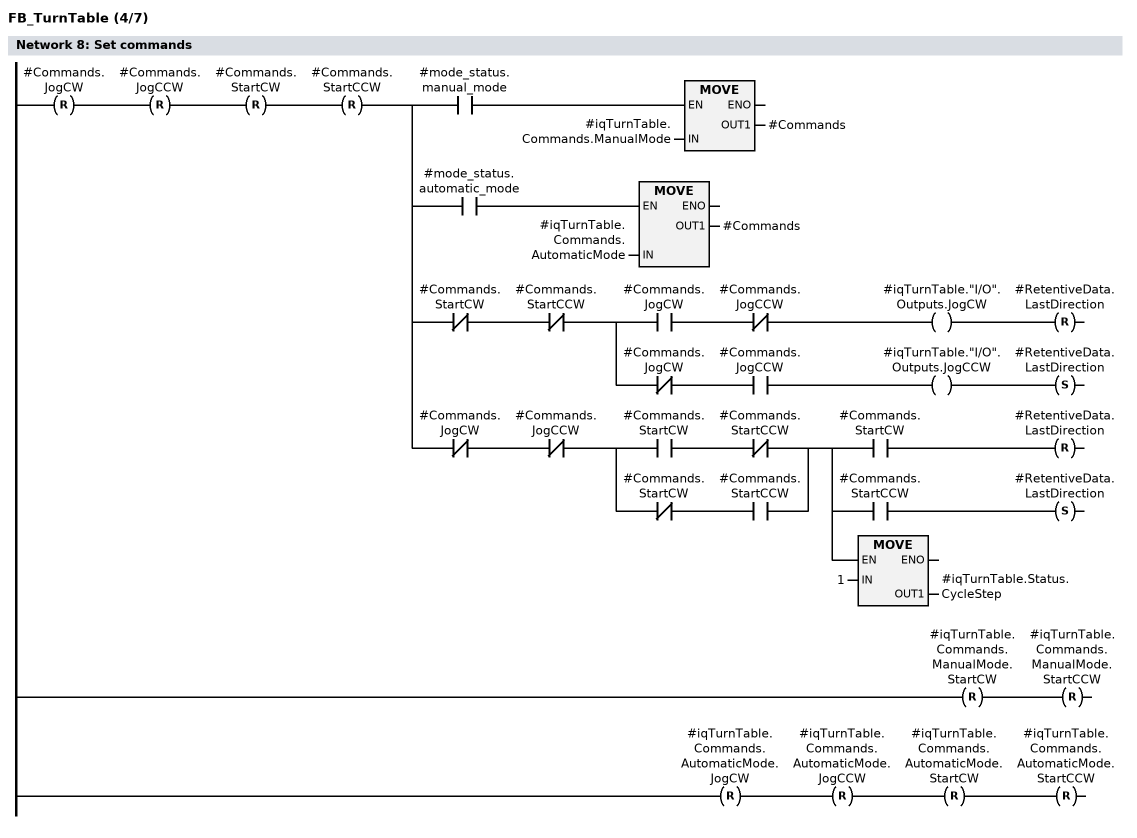
   RUNG wire#powerrail
      R_Coil( #Commands.JogCW )
      R_Coil( #Commands.JogCCW )
      R_Coil( #Commands.StartCW )
      R_Coil( #Commands.StartCCW )
      wire#w1
      Contact( #mode_status.manual_mode )
      Move(in := #iqTurnTable.Commands.ManualMode, out1 => #Commands)
   END_RUNG
   RUNG wire#w1
      Contact( #mode_status.automatic_mode )
      Move(in := #iqTurnTable.Commands.AutomaticMode, out1 => #Commands)
   END_RUNG
   RUNG wire#w1
      I_Contact( #Commands.StartCW )
      I_Contact( #Commands.StartCCW )
      wire#w2
      Contact( #Commands.JogCW )
      I_Contact( #Commands.JogCCW )
      Coil( #iqTurnTable."I/O".Outputs.JogCW )
      R_Coil( #RetentiveData.LastDirection )
   END_RUNG
   RUNG wire#w2
      I_Contact( #Commands.JogCW )
      Contact( #Commands.JogCCW )
      Coil( #iqTurnTable."I/O".Outputs.JogCCW )
      S_Coil( #RetentiveData.LastDirection )
   END_RUNG
   RUNG wire#w1
      I_Contact( #Commands.JogCW )
      I_Contact( #Commands.JogCCW )
      wire#w3
      Contact( #Commands.StartCW )
      I_Contact( #Commands.StartCCW )
      wire#w4
      Contact( #Commands.StartCW )
      R_Coil( #RetentiveData.LastDirection )
   END_RUNG
   RUNG wire#w3
      I_Contact( #Commands.StartCW )
      Contact( #Commands.StartCCW )
   END_RUNG wire#w4
   RUNG wire#w4
      Contact( #Commands.StartCCW )
      S_Coil( #RetentiveData.LastDirection )
   END_RUNG
   RUNG wire#w4
      Move(in := 1, out1 => #iqTurnTable.Status.CycleStep)
   END_RUNG
   RUNG wire#powerrail
      R_Coil( #iqTurnTable.Commands.ManualMode.StartCW )
      R_Coil( #iqTurnTable.Commands.ManualMode.StartCCW )
   END_RUNG
   RUNG wire#powerrail
      R_Coil( #iqTurnTable.Commands.AutomaticMode.JogCW )
      R_Coil( #iqTurnTable.Commands.AutomaticMode.JogCCW )
      R_Coil( #iqTurnTable.Commands.AutomaticMode.StartCW )
      R_Coil( #iqTurnTable.Commands.AutomaticMode.StartCCW )
   END_RUNG
   // the same network as SCL:
   #Commands.JogCW := FALSE;
   #Commands.JogCCW := FALSE;
   #Commands.StartCW := FALSE;
   #Commands.StartCCW := FALSE;
   IF #mode_status.manual_mode THEN #Commands := #iqTurnTable.Commands.ManualMode; END_IF;
   IF #mode_status.automatic_mode THEN #Commands := #iqTurnTable.Commands.AutomaticMode; END_IF;
   #_w1 := NOT #Commands.StartCW AND NOT #Commands.StartCCW;
   #iqTurnTable."I/O".Outputs.JogCW := #_w1 AND #Commands.JogCW AND NOT #Commands.JogCCW;
   IF #iqTurnTable."I/O".Outputs.JogCW THEN #RetentiveData.LastDirection := FALSE; END_IF;
   #iqTurnTable."I/O".Outputs.JogCCW := #_w1 AND NOT #Commands.JogCW AND #Commands.JogCCW;
   IF #iqTurnTable."I/O".Outputs.JogCCW THEN #RetentiveData.LastDirection := TRUE; END_IF;
   #_w2 := NOT #Commands.JogCW AND NOT #Commands.JogCCW AND ((#Commands.StartCW AND NOT #Commands.StartCCW) OR (NOT #Commands.StartCW AND #Commands.StartCCW));
   IF #_w2 AND #Commands.StartCW THEN #RetentiveData.LastDirection := FALSE; END_IF;
   IF #_w2 AND #Commands.StartCCW THEN #RetentiveData.LastDirection := TRUE; END_IF;
   IF #_w2 THEN #iqTurnTable.Status.CycleStep := 1; END_IF;
   #iqTurnTable.Commands.ManualMode.StartCW := FALSE;
   #iqTurnTable.Commands.ManualMode.StartCCW := FALSE;
   #iqTurnTable.Commands.AutomaticMode.JogCW := FALSE;
   #iqTurnTable.Commands.AutomaticMode.JogCCW := FALSE;
   #iqTurnTable.Commands.AutomaticMode.StartCW := FALSE;
   #iqTurnTable.Commands.AutomaticMode.StartCCW := FALSE;
END_REGION

REGION Network 9: Cycle: Reset
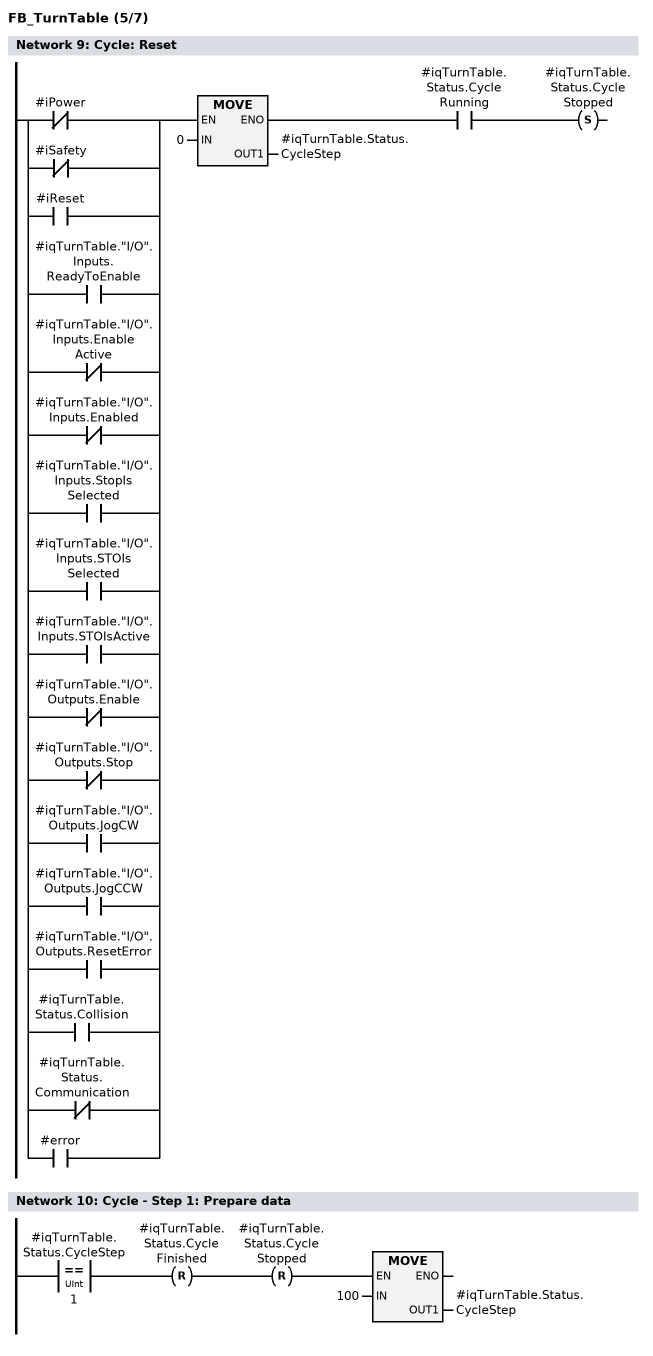
   RUNG wire#powerrail
      I_Contact( #iPower )
      wire#w1
      Move(in := 0, out1 => #iqTurnTable.Status.CycleStep)
      Contact( #iqTurnTable.Status.CycleRunning )
      S_Coil( #iqTurnTable.Status.CycleStopped )
   END_RUNG
   RUNG wire#powerrail
      I_Contact( #iSafety )
   END_RUNG wire#w1
   RUNG wire#powerrail
      Contact( #iReset )
   END_RUNG wire#w1
   RUNG wire#powerrail
      Contact( #iqTurnTable."I/O".Inputs.ReadyToEnable )
   END_RUNG wire#w1
   RUNG wire#powerrail
      I_Contact( #iqTurnTable."I/O".Inputs.EnableActive )
   END_RUNG wire#w1
   RUNG wire#powerrail
      I_Contact( #iqTurnTable."I/O".Inputs.Enabled )
   END_RUNG wire#w1
   RUNG wire#powerrail
      Contact( #iqTurnTable."I/O".Inputs.StopIsSelected )
   END_RUNG wire#w1
   RUNG wire#powerrail
      Contact( #iqTurnTable."I/O".Inputs.STOIsSelected )
   END_RUNG wire#w1
   RUNG wire#powerrail
      Contact( #iqTurnTable."I/O".Inputs.STOIsActive )
   END_RUNG wire#w1
   RUNG wire#powerrail
      I_Contact( #iqTurnTable."I/O".Outputs.Enable )
   END_RUNG wire#w1
   RUNG wire#powerrail
      I_Contact( #iqTurnTable."I/O".Outputs.Stop )
   END_RUNG wire#w1
   RUNG wire#powerrail
      Contact( #iqTurnTable."I/O".Outputs.JogCW )
   END_RUNG wire#w1
   RUNG wire#powerrail
      Contact( #iqTurnTable."I/O".Outputs.JogCCW )
   END_RUNG wire#w1
   RUNG wire#powerrail
      Contact( #iqTurnTable."I/O".Outputs.ResetError )
   END_RUNG wire#w1
   RUNG wire#powerrail
      Contact( #iqTurnTable.Status.Collision )
   END_RUNG wire#w1
   RUNG wire#powerrail
      I_Contact( #iqTurnTable.Status.Communication )
   END_RUNG wire#w1
   RUNG wire#powerrail
      Contact( #error )
   END_RUNG wire#w1
   // the same network as SCL:
   #_w1 := NOT #iPower OR NOT #iSafety OR #iReset OR #iqTurnTable."I/O".Inputs.ReadyToEnable OR NOT #iqTurnTable."I/O".Inputs.EnableActive OR NOT #iqTurnTable."I/O".Inputs.Enabled OR #iqTurnTable."I/O".Inputs.StopIsSelected OR #iqTurnTable."I/O".Inputs.STOIsSelected OR #iqTurnTable."I/O".Inputs.STOIsActive OR NOT #iqTurnTable."I/O".Outputs.Enable OR NOT #iqTurnTable."I/O".Outputs.Stop OR #iqTurnTable."I/O".Outputs.JogCW OR #iqTurnTable."I/O".Outputs.JogCCW OR #iqTurnTable."I/O".Outputs.ResetError OR #iqTurnTable.Status.Collision OR NOT #iqTurnTable.Status.Communication OR #error;
   IF #_w1 THEN #iqTurnTable.Status.CycleStep := 0; END_IF;
   IF #_w1 AND #iqTurnTable.Status.CycleRunning THEN #iqTurnTable.Status.CycleStopped := TRUE; END_IF;
END_REGION

REGION Network 10: Cycle - Step 1: Prepare data
   RUNG wire#powerrail
      { S7_Templates := "SrcType := UInt" } EQ_Contact(in1 := #iqTurnTable.Status.CycleStep, in2 := 1)
      R_Coil( #iqTurnTable.Status.CycleFinished )
      R_Coil( #iqTurnTable.Status.CycleStopped )
      Move(in := 100, out1 => #iqTurnTable.Status.CycleStep)
   END_RUNG
   // the same network as SCL:
   IF #iqTurnTable.Status.CycleStep = 1 THEN
       #iqTurnTable.Status.CycleFinished := FALSE;
       #iqTurnTable.Status.CycleStopped := FALSE;
       #iqTurnTable.Status.CycleStep := 100;
   END_IF;
END_REGION

REGION Network 11: Cycle - Step 100: Check out of position
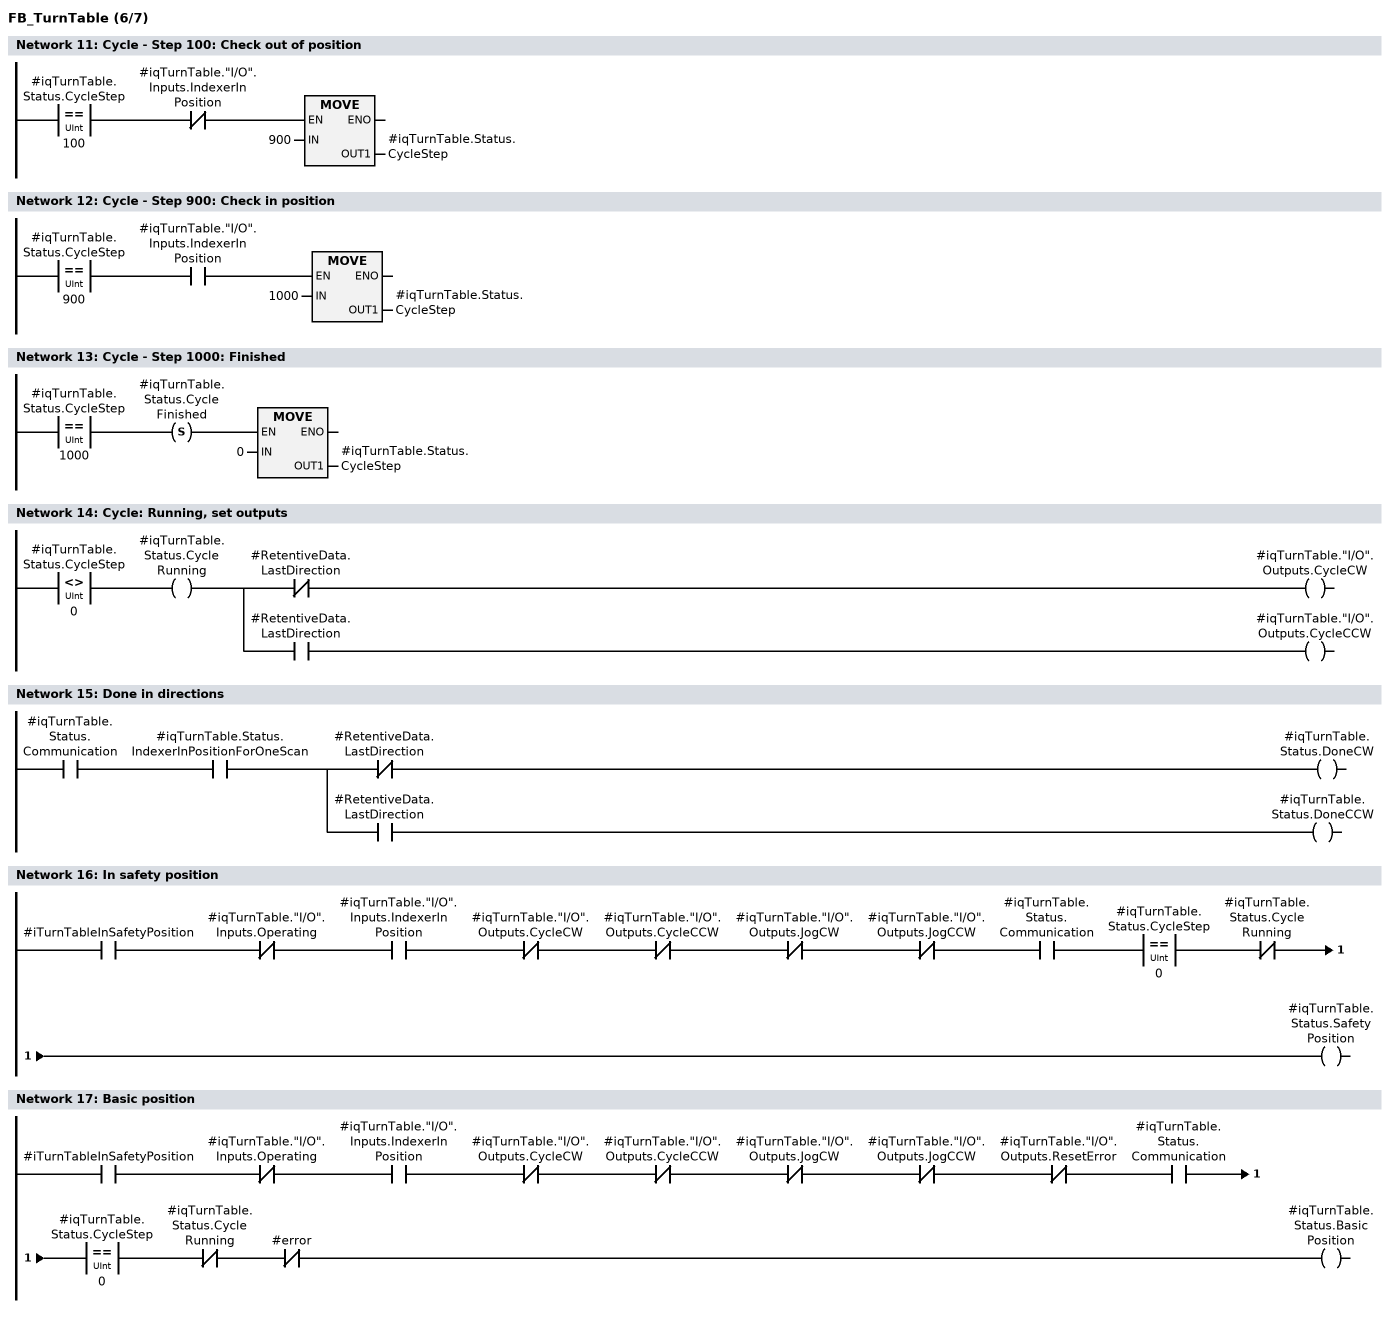
   RUNG wire#powerrail
      { S7_Templates := "SrcType := UInt" } EQ_Contact(in1 := #iqTurnTable.Status.CycleStep, in2 := 100)
      I_Contact( #iqTurnTable."I/O".Inputs.IndexerInPosition )
      Move(in := 900, out1 => #iqTurnTable.Status.CycleStep)
   END_RUNG
   // the same network as SCL:
   IF (#iqTurnTable.Status.CycleStep = 100) AND NOT #iqTurnTable."I/O".Inputs.IndexerInPosition THEN
       #iqTurnTable.Status.CycleStep := 900;
   END_IF;
END_REGION

REGION Network 12: Cycle - Step 900: Check in position
   RUNG wire#powerrail
      { S7_Templates := "SrcType := UInt" } EQ_Contact(in1 := #iqTurnTable.Status.CycleStep, in2 := 900)
      Contact( #iqTurnTable."I/O".Inputs.IndexerInPosition )
      Move(in := 1000, out1 => #iqTurnTable.Status.CycleStep)
   END_RUNG
   // the same network as SCL:
   IF (#iqTurnTable.Status.CycleStep = 900) AND #iqTurnTable."I/O".Inputs.IndexerInPosition THEN
       #iqTurnTable.Status.CycleStep := 1000;
   END_IF;
END_REGION

REGION Network 13: Cycle - Step 1000: Finished
   RUNG wire#powerrail
      { S7_Templates := "SrcType := UInt" } EQ_Contact(in1 := #iqTurnTable.Status.CycleStep, in2 := 1000)
      S_Coil( #iqTurnTable.Status.CycleFinished )
      Move(in := 0, out1 => #iqTurnTable.Status.CycleStep)
   END_RUNG
   // the same network as SCL:
   IF #iqTurnTable.Status.CycleStep = 1000 THEN
       #iqTurnTable.Status.CycleFinished := TRUE;
       #iqTurnTable.Status.CycleStep := 0;
   END_IF;
END_REGION

REGION Network 14: Cycle: Running, set outputs
   RUNG wire#powerrail
      { S7_Templates := "SrcType := UInt" } NE_Contact(in1 := #iqTurnTable.Status.CycleStep, in2 := 0)
      Coil( #iqTurnTable.Status.CycleRunning )
      wire#w1
      I_Contact( #RetentiveData.LastDirection )
      Coil( #iqTurnTable."I/O".Outputs.CycleCW )
   END_RUNG
   RUNG wire#w1
      Contact( #RetentiveData.LastDirection )
      Coil( #iqTurnTable."I/O".Outputs.CycleCCW )
   END_RUNG
   // the same network as SCL:
   #iqTurnTable.Status.CycleRunning := #iqTurnTable.Status.CycleStep <> 0;
   #iqTurnTable."I/O".Outputs.CycleCW := #iqTurnTable.Status.CycleRunning AND NOT #RetentiveData.LastDirection;
   #iqTurnTable."I/O".Outputs.CycleCCW := #iqTurnTable.Status.CycleRunning AND #RetentiveData.LastDirection;
END_REGION

REGION Network 15: Done in directions
   RUNG wire#powerrail
      Contact( #iqTurnTable.Status.Communication )
      Contact( #iqTurnTable.Status.IndexerInPositionForOneScan )
      wire#w1
      I_Contact( #RetentiveData.LastDirection )
      Coil( #iqTurnTable.Status.DoneCW )
   END_RUNG
   RUNG wire#w1
      Contact( #RetentiveData.LastDirection )
      Coil( #iqTurnTable.Status.DoneCCW )
   END_RUNG
   // the same network as SCL:
   #_w1 := #iqTurnTable.Status.Communication AND #iqTurnTable.Status.IndexerInPositionForOneScan;
   #iqTurnTable.Status.DoneCW := #_w1 AND NOT #RetentiveData.LastDirection;
   #iqTurnTable.Status.DoneCCW := #_w1 AND #RetentiveData.LastDirection;
END_REGION

REGION Network 16: In safety position
   RUNG wire#powerrail
      Contact( #iTurnTableInSafetyPosition )
      I_Contact( #iqTurnTable."I/O".Inputs.Operating )
      Contact( #iqTurnTable."I/O".Inputs.IndexerInPosition )
      I_Contact( #iqTurnTable."I/O".Outputs.CycleCW )
      I_Contact( #iqTurnTable."I/O".Outputs.CycleCCW )
      I_Contact( #iqTurnTable."I/O".Outputs.JogCW )
      I_Contact( #iqTurnTable."I/O".Outputs.JogCCW )
      Contact( #iqTurnTable.Status.Communication )
      { S7_Templates := "SrcType := UInt" } EQ_Contact(in1 := #iqTurnTable.Status.CycleStep, in2 := 0)
      I_Contact( #iqTurnTable.Status.CycleRunning )
      Coil( #iqTurnTable.Status.SafetyPosition )
   END_RUNG
   // the same network as SCL:
   #iqTurnTable.Status.SafetyPosition := #iTurnTableInSafetyPosition AND NOT #iqTurnTable."I/O".Inputs.Operating AND #iqTurnTable."I/O".Inputs.IndexerInPosition AND NOT #iqTurnTable."I/O".Outputs.CycleCW AND NOT #iqTurnTable."I/O".Outputs.CycleCCW AND NOT #iqTurnTable."I/O".Outputs.JogCW AND NOT #iqTurnTable."I/O".Outputs.JogCCW AND #iqTurnTable.Status.Communication AND (#iqTurnTable.Status.CycleStep = 0) AND NOT #iqTurnTable.Status.CycleRunning;
END_REGION

REGION Network 17: Basic position
   RUNG wire#powerrail
      Contact( #iTurnTableInSafetyPosition )
      I_Contact( #iqTurnTable."I/O".Inputs.Operating )
      Contact( #iqTurnTable."I/O".Inputs.IndexerInPosition )
      I_Contact( #iqTurnTable."I/O".Outputs.CycleCW )
      I_Contact( #iqTurnTable."I/O".Outputs.CycleCCW )
      I_Contact( #iqTurnTable."I/O".Outputs.JogCW )
      I_Contact( #iqTurnTable."I/O".Outputs.JogCCW )
      I_Contact( #iqTurnTable."I/O".Outputs.ResetError )
      Contact( #iqTurnTable.Status.Communication )
      { S7_Templates := "SrcType := UInt" } EQ_Contact(in1 := #iqTurnTable.Status.CycleStep, in2 := 0)
      I_Contact( #iqTurnTable.Status.CycleRunning )
      I_Contact( #error )
      Coil( #iqTurnTable.Status.BasicPosition )
   END_RUNG
   // the same network as SCL:
   #iqTurnTable.Status.BasicPosition := #iTurnTableInSafetyPosition AND NOT #iqTurnTable."I/O".Inputs.Operating AND #iqTurnTable."I/O".Inputs.IndexerInPosition AND NOT #iqTurnTable."I/O".Outputs.CycleCW AND NOT #iqTurnTable."I/O".Outputs.CycleCCW AND NOT #iqTurnTable."I/O".Outputs.JogCW AND NOT #iqTurnTable."I/O".Outputs.JogCCW AND NOT #iqTurnTable."I/O".Outputs.ResetError AND #iqTurnTable.Status.Communication AND (#iqTurnTable.Status.CycleStep = 0) AND NOT #iqTurnTable.Status.CycleRunning AND NOT #error;
END_REGION

REGION Network 18: Set outputs
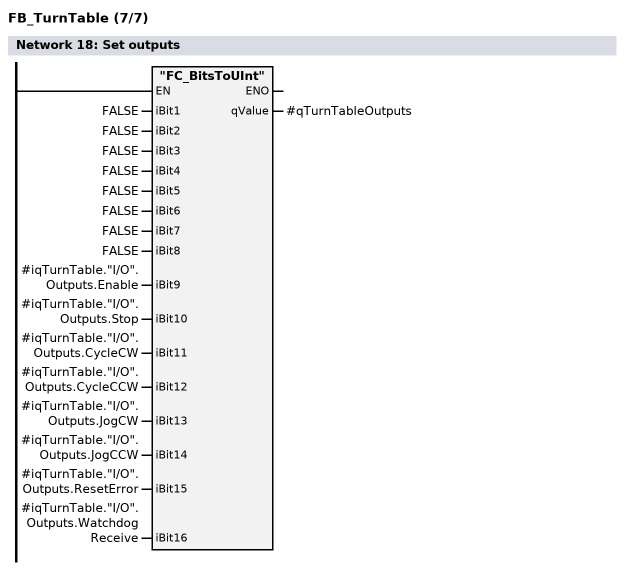
   RUNG wire#powerrail
      "FC_BitsToUInt"(iBit1 := FALSE, iBit2 := FALSE, iBit3 := FALSE, iBit4 := FALSE, iBit5 := FALSE, iBit6 := FALSE, iBit7 := FALSE, iBit8 := FALSE, iBit9 := #iqTurnTable."I/O".Outputs.Enable, iBit10 := #iqTurnTable."I/O".Outputs.Stop, iBit11 := #iqTurnTable."I/O".Outputs.CycleCW, iBit12 := #iqTurnTable."I/O".Outputs.CycleCCW, iBit13 := #iqTurnTable."I/O".Outputs.JogCW, iBit14 := #iqTurnTable."I/O".Outputs.JogCCW, iBit15 := #iqTurnTable."I/O".Outputs.ResetError, iBit16 := #iqTurnTable."I/O".Outputs.WatchdogReceive, qValue => #qTurnTableOutputs)
   END_RUNG
   // the same network as SCL:
   "FC_BitsToUInt"(iBit1 := FALSE,
                   iBit2 := FALSE,
                   iBit3 := FALSE,
                   iBit4 := FALSE,
                   iBit5 := FALSE,
                   iBit6 := FALSE,
                   iBit7 := FALSE,
                   iBit8 := FALSE,
                   iBit9 := #iqTurnTable."I/O".Outputs.Enable,
                   iBit10 := #iqTurnTable."I/O".Outputs.Stop,
                   iBit11 := #iqTurnTable."I/O".Outputs.CycleCW,
                   iBit12 := #iqTurnTable."I/O".Outputs.CycleCCW,
                   iBit13 := #iqTurnTable."I/O".Outputs.JogCW,
                   iBit14 := #iqTurnTable."I/O".Outputs.JogCCW,
                   iBit15 := #iqTurnTable."I/O".Outputs.ResetError,
                   iBit16 := #iqTurnTable."I/O".Outputs.WatchdogReceive,
                   qValue => #qTurnTableOutputs);
END_REGION
END_FUNCTION_BLOCK

FUNCTION "FC_UIntToBits" : Void   // FC1021, LAD
{ S7_Optimized_Access := 'FALSE' }
VERSION : 0.1
// stored: AutoNumber false, IsIECCheckEnabled false, SetENOAutomatically false, UDAEnableTagReadback false
   VAR_INPUT
      iValue : UInt;
   END_VAR
   VAR_OUTPUT
      qBit1 : Bool;
      qBit2 : Bool;
      qBit3 : Bool;
      qBit4 : Bool;
      qBit5 : Bool;
      qBit6 : Bool;
      qBit7 : Bool;
      qBit8 : Bool;
      qBit9 : Bool;
      qBit10 : Bool;
      qBit11 : Bool;
      qBit12 : Bool;
      qBit13 : Bool;
      qBit14 : Bool;
      qBit15 : Bool;
      qBit16 : Bool;
   END_VAR
   VAR_TEMP
      value : UInt;
   END_VAR
BEGIN

REGION Network 1: Convert UInt to bits
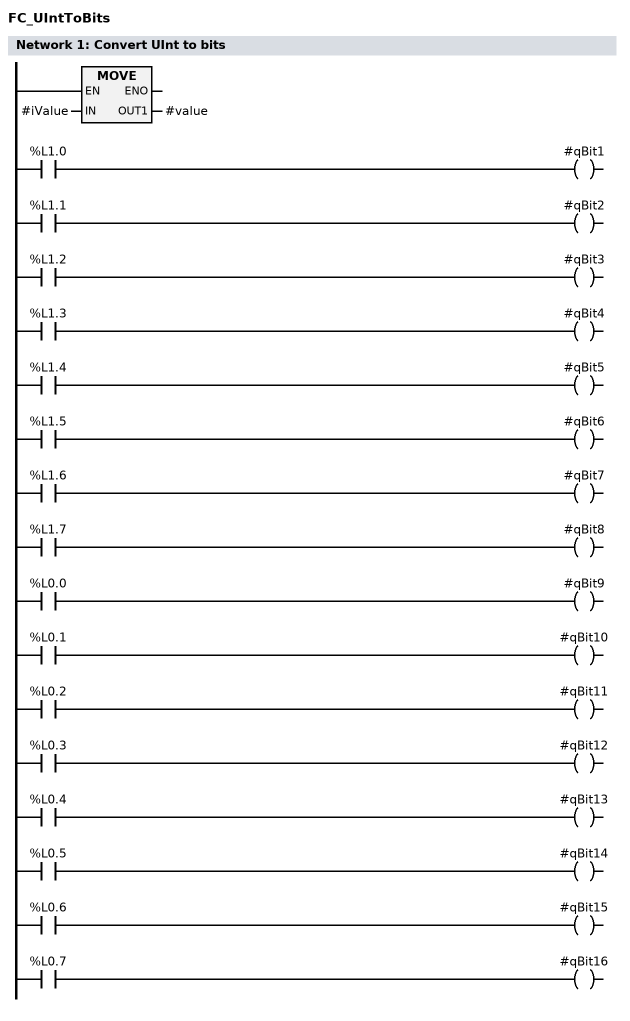
   RUNG wire#powerrail
      Move(in := #iValue, out1 => #value)
   END_RUNG
   RUNG wire#powerrail
      Contact( %L1.0 )
      Coil( #qBit1 )
   END_RUNG
   RUNG wire#powerrail
      Contact( %L1.1 )
      Coil( #qBit2 )
   END_RUNG
   RUNG wire#powerrail
      Contact( %L1.2 )
      Coil( #qBit3 )
   END_RUNG
   RUNG wire#powerrail
      Contact( %L1.3 )
      Coil( #qBit4 )
   END_RUNG
   RUNG wire#powerrail
      Contact( %L1.4 )
      Coil( #qBit5 )
   END_RUNG
   RUNG wire#powerrail
      Contact( %L1.5 )
      Coil( #qBit6 )
   END_RUNG
   RUNG wire#powerrail
      Contact( %L1.6 )
      Coil( #qBit7 )
   END_RUNG
   RUNG wire#powerrail
      Contact( %L1.7 )
      Coil( #qBit8 )
   END_RUNG
   RUNG wire#powerrail
      Contact( %L0.0 )
      Coil( #qBit9 )
   END_RUNG
   RUNG wire#powerrail
      Contact( %L0.1 )
      Coil( #qBit10 )
   END_RUNG
   RUNG wire#powerrail
      Contact( %L0.2 )
      Coil( #qBit11 )
   END_RUNG
   RUNG wire#powerrail
      Contact( %L0.3 )
      Coil( #qBit12 )
   END_RUNG
   RUNG wire#powerrail
      Contact( %L0.4 )
      Coil( #qBit13 )
   END_RUNG
   RUNG wire#powerrail
      Contact( %L0.5 )
      Coil( #qBit14 )
   END_RUNG
   RUNG wire#powerrail
      Contact( %L0.6 )
      Coil( #qBit15 )
   END_RUNG
   RUNG wire#powerrail
      Contact( %L0.7 )
      Coil( #qBit16 )
   END_RUNG
   // the same network as SCL:
   #value := #iValue;
   #qBit1 := %L1.0;
   #qBit2 := %L1.1;
   #qBit3 := %L1.2;
   #qBit4 := %L1.3;
   #qBit5 := %L1.4;
   #qBit6 := %L1.5;
   #qBit7 := %L1.6;
   #qBit8 := %L1.7;
   #qBit9 := %L0.0;
   #qBit10 := %L0.1;
   #qBit11 := %L0.2;
   #qBit12 := %L0.3;
   #qBit13 := %L0.4;
   #qBit14 := %L0.5;
   #qBit15 := %L0.6;
   #qBit16 := %L0.7;
END_REGION
END_FUNCTION

FUNCTION "FC_BitsToUInt" : Void   // FC1020, LAD
{ S7_Optimized_Access := 'FALSE' }
VERSION : 0.1
// stored: AutoNumber false, IsIECCheckEnabled false, SetENOAutomatically false, UDAEnableTagReadback false
   VAR_INPUT
      iBit1 : Bool;
      iBit2 : Bool;
      iBit3 : Bool;
      iBit4 : Bool;
      iBit5 : Bool;
      iBit6 : Bool;
      iBit7 : Bool;
      iBit8 : Bool;
      iBit9 : Bool;
      iBit10 : Bool;
      iBit11 : Bool;
      iBit12 : Bool;
      iBit13 : Bool;
      iBit14 : Bool;
      iBit15 : Bool;
      iBit16 : Bool;
   END_VAR
   VAR_OUTPUT
      qValue : UInt;
   END_VAR
   VAR_TEMP
      value : UInt;
   END_VAR
BEGIN

REGION Network 1: Convert bits to UInt
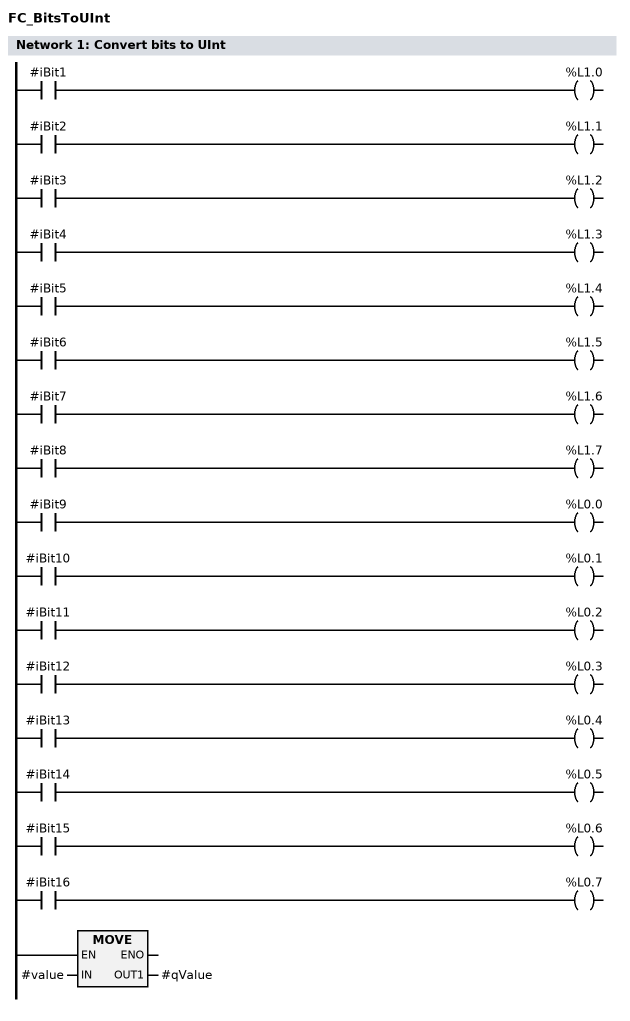
   RUNG wire#powerrail
      Contact( #iBit1 )
      Coil( %L1.0 )
   END_RUNG
   RUNG wire#powerrail
      Contact( #iBit2 )
      Coil( %L1.1 )
   END_RUNG
   RUNG wire#powerrail
      Contact( #iBit3 )
      Coil( %L1.2 )
   END_RUNG
   RUNG wire#powerrail
      Contact( #iBit4 )
      Coil( %L1.3 )
   END_RUNG
   RUNG wire#powerrail
      Contact( #iBit5 )
      Coil( %L1.4 )
   END_RUNG
   RUNG wire#powerrail
      Contact( #iBit6 )
      Coil( %L1.5 )
   END_RUNG
   RUNG wire#powerrail
      Contact( #iBit7 )
      Coil( %L1.6 )
   END_RUNG
   RUNG wire#powerrail
      Contact( #iBit8 )
      Coil( %L1.7 )
   END_RUNG
   RUNG wire#powerrail
      Contact( #iBit9 )
      Coil( %L0.0 )
   END_RUNG
   RUNG wire#powerrail
      Contact( #iBit10 )
      Coil( %L0.1 )
   END_RUNG
   RUNG wire#powerrail
      Contact( #iBit11 )
      Coil( %L0.2 )
   END_RUNG
   RUNG wire#powerrail
      Contact( #iBit12 )
      Coil( %L0.3 )
   END_RUNG
   RUNG wire#powerrail
      Contact( #iBit13 )
      Coil( %L0.4 )
   END_RUNG
   RUNG wire#powerrail
      Contact( #iBit14 )
      Coil( %L0.5 )
   END_RUNG
   RUNG wire#powerrail
      Contact( #iBit15 )
      Coil( %L0.6 )
   END_RUNG
   RUNG wire#powerrail
      Contact( #iBit16 )
      Coil( %L0.7 )
   END_RUNG
   RUNG wire#powerrail
      Move(in := #value, out1 => #qValue)
   END_RUNG
   // the same network as SCL:
   %L1.0 := #iBit1;
   %L1.1 := #iBit2;
   %L1.2 := #iBit3;
   %L1.3 := #iBit4;
   %L1.4 := #iBit5;
   %L1.5 := #iBit6;
   %L1.6 := #iBit7;
   %L1.7 := #iBit8;
   %L0.0 := #iBit9;
   %L0.1 := #iBit10;
   %L0.2 := #iBit11;
   %L0.3 := #iBit12;
   %L0.4 := #iBit13;
   %L0.5 := #iBit14;
   %L0.6 := #iBit15;
   %L0.7 := #iBit16;
   #qValue := #value;
END_REGION
END_FUNCTION

FUNCTION_BLOCK "CycleTimeMeas"   // FB46, FBD
{ S7_Optimized_Access := 'FALSE' }
VERSION : 0.1
// stored: AutoNumber false, IsIECCheckEnabled false, SetENOAutomatically false, UDAEnableTagReadback false
   VAR_INPUT
      StartCycle : Bool;
      ResetHistory : Bool;
   END_VAR
   VAR DB_SPECIFIC
      ActualTime : Time;
      LastTime : Time;
      edge2 : Bool;
      edge1 : Bool;
      Suma : DInt;
      Count : DInt;
      Max : Time;
      Min : Time;
      Average : Time;
      IEC_Timer_0_Instance { S7_SetPoint := 'True'} : TON_TIME;
      History : Array[1..20] of Time;
      NewTime : Bool;
   END_VAR
   VAR_TEMP
      d : DInt;
      i : Int;
   END_VAR
   VAR_TEMP   // added for the SCL form of the ladder/FBD networks
      _w1 : Bool;
   END_VAR
BEGIN

NETWORK
TITLE = Convert time to dint
      L     #ActualTime;
      T     #d;


REGION Network 2: Save cycle time
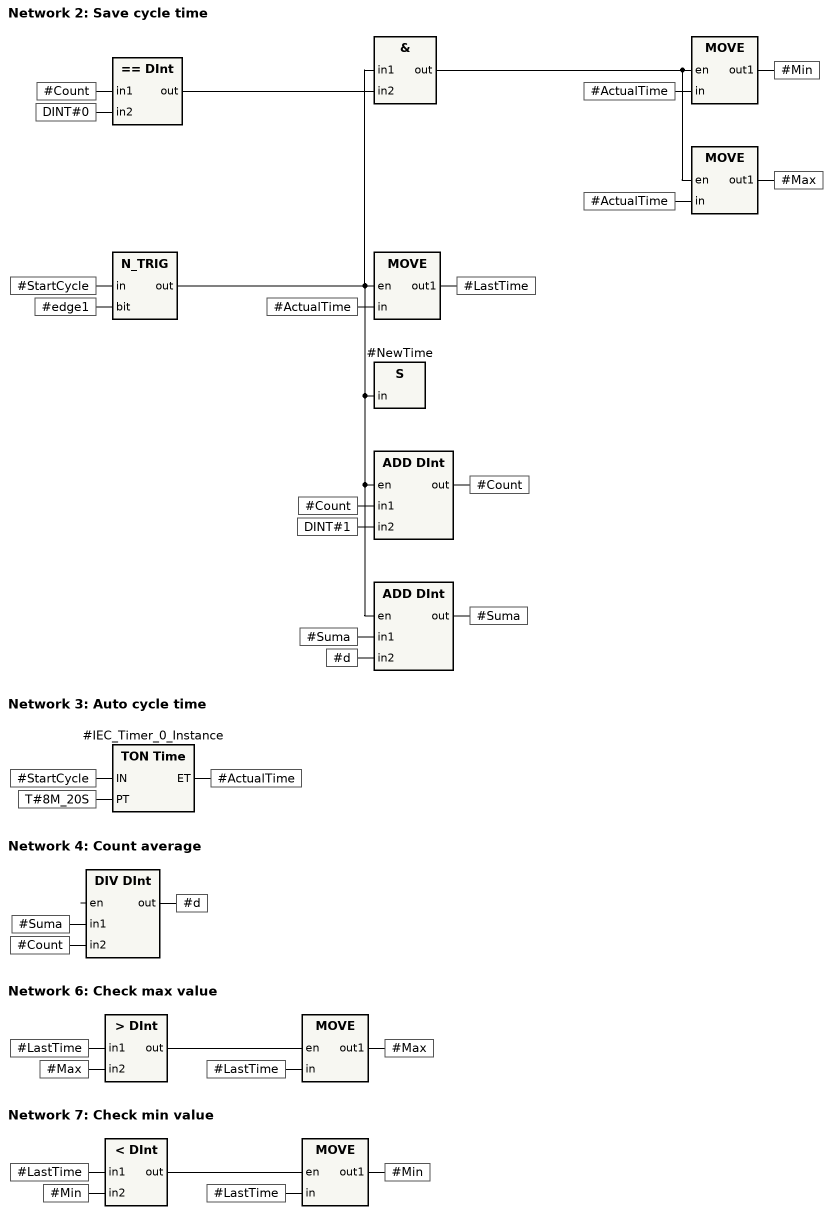
   #_w1 := NOT #StartCycle AND #edge1;   // falling edge
   #edge1 := #StartCycle;
   IF #_w1 THEN
       #LastTime := #ActualTime;
       #NewTime := TRUE;
   END_IF;
   IF #_w1 AND (#Count = DINT#0) THEN
       #Min := #ActualTime;
       #Max := #ActualTime;
   END_IF;
   IF #_w1 THEN
       #Count := #Count + DINT#1;
       #Suma := #Suma + #d;
   END_IF;
END_REGION

REGION Network 3: Auto cycle time
   #IEC_Timer_0_Instance(IN := #StartCycle, PT := T#8M_20S, ET => #ActualTime);   // TON
END_REGION

REGION Network 4: Count average
   #d := #Suma / #Count;
END_REGION

NETWORK
TITLE = Convert dint to time
      L     #d;
      T     #Average;


REGION Network 6: Check max value
   IF #LastTime > #Max THEN #Max := #LastTime; END_IF;
END_REGION

REGION Network 7: Check min value
   IF #LastTime < #Min THEN #Min := #LastTime; END_IF;
END_REGION

REGION Network 8: Reset history
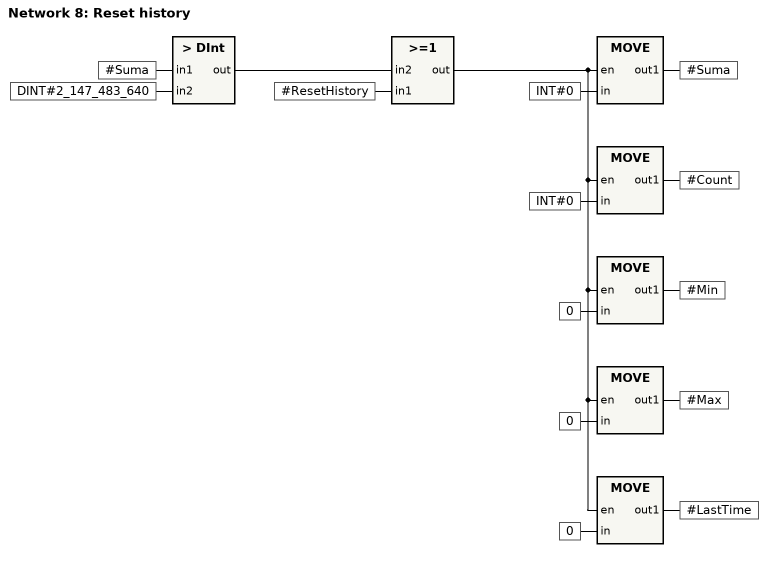
   #_w1 := (#Suma > DINT#2_147_483_640) OR #ResetHistory;
   IF #_w1 THEN
       #Suma := INT#0;
       #Count := INT#0;
       #Min := 0;
       #Max := 0;
       #LastTime := 0;
   END_IF;
END_REGION

REGION Network 10 (SCL)
   IF #NewTime THEN
       FOR #i := 1 TO 19 DO
           #History[21 - #i] := #History[20 - #i];
       END_FOR;
       #History[1] := #LastTime;
   END_IF;
   #NewTime := false;
END_REGION
END_FUNCTION_BLOCK

FUNCTION_BLOCK "RobotMain"
{ S7_Optimized_Access := 'TRUE' }
VERSION : 0.1
   VAR_OUTPUT 
      RobotInStartingPosition : Bool;
   END_VAR

   VAR 
      R1 : "RobotControl";
      R_TRIG_Instance {InstructionName := 'R_TRIG'; LibVersion := '1.0'} : R_TRIG;
      F_TRIG_Instance {InstructionName := 'F_TRIG'; LibVersion := '1.0'} : F_TRIG;
   END_VAR


BEGIN
	REGION cylinders positions
	    "qR1_MM220grippingTubeInBp" := "DevicesData".Cylinders["MM2200_GrippingTubeFront"].InBp;
	    "qR1_MM220grippingTubeInWp" := "DevicesData".Cylinders["MM2200_GrippingTubeFront"].InWp;
	    "qR1_MM222holdingSidememberInsideInBp" := "DevicesData".Cylinders["MM2220_HoldingSidememberInsideLeft"].InBp;
	    "qR1_MM222holdingSidememberInsideInWp" := "DevicesData".Cylinders["MM2220_HoldingSidememberInsideLeft"].InWp;
	    "qR1_MM224holdingSidememberOutsideInBp" := "DevicesData".Cylinders["MM2240_HoldingSidememberOutsideLeft"].InBp;
	    "qR1_MM224holdingSidememberOutsideInWp" := "DevicesData".Cylinders["MM2240_HoldingSidememberOutsideLeft"].InWp;
	END_REGION
	REGION cylinders control in automat 
	    IF "ModeSelection_DB".mode.activeMode = "mode_2_base" OR
	        "ModeSelection_DB".mode.activeMode = "mode_3_automat" OR
	        "ModeSelection_DB".mode.activeMode = "mode_4_semiautomat"
	    THEN
	        "DevicesData".Cylinders["MM2200_GrippingTubeFront"].ToBp := "iR1_MM220grippingTubeToBp";
	        "DevicesData".Cylinders["MM2200_GrippingTubeFront"].ToWp := "iR1_MM220grippingTubeToWp";
	        "DevicesData".Cylinders["MM2220_HoldingSidememberInsideLeft"].ToBp := "iR1_MM222holdingSidememberInsideToBp";
	        "DevicesData".Cylinders["MM2220_HoldingSidememberInsideLeft"].ToWp := "iR1_MM222holdingSidememberInsideToWp";
	        "DevicesData".Cylinders["MM2240_HoldingSidememberOutsideLeft"].ToBp := "iR1_MM224holdingSidememberOutsideToBp";
	        "DevicesData".Cylinders["MM2240_HoldingSidememberOutsideLeft"].ToWp := "iR1_MM224holdingSidememberOutsideToWp";
	    END_IF;
	 END_REGION
	REGION part present
	    "qR1frontTubePresent" := "iR1tubePresentFront";
	    "qR1rearTubePresent" := "iR1tubePresentRear";
	END_REGION
	REGION type
	    "qR1typeRH" := "DB_ProductionProgramActual".Program.MechanicalType = 1;
	END_REGION
	
	"RobotJob_DB"(OFF_SQ := NOT "DevicesData".R1.Job.Start,
	               INIT_SQ := "DevicesData".R1.Job.Start,
	               ACK_EF:="Alarms".Reset);
	 
	"DevicesData".R1.StartReq := ("SystemHMI".AutomaticMode OR "SystemHMI".GoToBasicPosition) AND "safety_signals"."4L+";
	#R1(StartReq := "DevicesData".R1.StartReq,
	    KeyExt := "DevicesData".R1.StartReq,
	    JobNrReq := "DevicesData".R1.Job.JobNr,
	    periReady := "iR1periReady",
	    stopMess := "iR1stopMess",
	    progAct := "iR1progAct",
	    onPath := "iR1onPath",
	    ext := "iR1ext",
	    internalEstop := "iR1internalEstop",
	    home := #RobotInStartingPosition,
	    pgNoReq := "iR1pgNoReq",
	    robStopped := "iR1robStopped",
	    jobNrBack := "iR1jobNr",
	    StartAllowed => "DevicesData".R1.StartAllowed,
	    Started => "DevicesData".R1.Started,
	    drivesOn => "qR1drivesOn",
	    confMess => "qR1confMess",
	    ExtStart => "qR1ExtStart",
	    reqHome => "qR1reqHome",
	    reqDoor => "qR1reqDoor",
	    jobNr => "qR1jobNr");
	
	"qR1moveEnable" :=
	("SystemHMI".AutomaticMode OR "SystemHMI".GoToBasicPosition) AND "safety_signals"."4L+" AND "iR1ext" OR
	NOT ("SystemHMI".AutomaticMode OR "SystemHMI".GoToBasicPosition) AND "safety_signals"."3L+" AND NOT "iR1ext";
	
	#RobotInStartingPosition :=
	"iR1home" OR
	"iR1inPickupStartPositionSt2" OR
	"iR1inDropoffStartPositionSt3" OR
	"iR1inPickupStartPositionAutoeject" OR
	"iR1inDropoffStartPositionHanger";
	
	
	
	
	
	
	
END_FUNCTION_BLOCK

FUNCTION_BLOCK "RobotControl"   // FB15, LAD
{ S7_Optimized_Access := 'TRUE' }
VERSION : 0.1
// stored: AutoNumber true, IsIECCheckEnabled false, IsRetainMemResEnabled false, MemoryReserve 100, SetENOAutomatically false, UDAEnableTagReadback false
   VAR_INPUT
      StartReq : Bool;
      KeyExt : Bool;
      JobNrReq : Byte;
      periReady : Bool;
      stopMess : Bool;
      progAct : Bool;
      onPath : Bool;
      ext : Bool;
      internalEstop : Bool;
      home : Bool;
      pgNoReq : Bool;
      robStopped : Bool;
      jobNrBack : Byte;
   END_VAR
   VAR_OUTPUT
      StartAllowed : Bool;
      Started : Bool;
      drivesOn : Bool;
      confMess : Bool;
      ExtStart : Bool;
      moveEnable : Bool;
      reqHome : Bool;
      pgNoValid : Bool;
      reqDoor : Bool;
      jobNr : Byte;
   END_VAR
BEGIN

REGION Network 1: Possible to start external auto
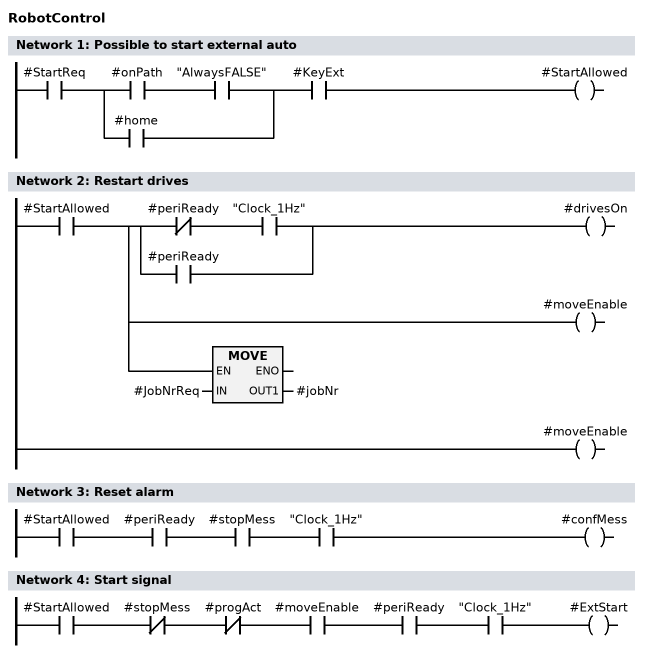
   RUNG wire#powerrail
      Contact( #StartReq )
      wire#w1
      Contact( #onPath )
      Contact( "AlwaysFALSE" )
      wire#w2
      Contact( #KeyExt )
      Coil( #StartAllowed )
   END_RUNG
   RUNG wire#w1
      Contact( #home )
   END_RUNG wire#w2
   // the same network as SCL:
   #StartAllowed := #StartReq AND ((#onPath AND "AlwaysFALSE") OR #home) AND #KeyExt;
END_REGION

REGION Network 2: Restart drives
   RUNG wire#powerrail
      Contact( #StartAllowed )
      wire#w1
      I_Contact( #periReady )
      Contact( "Clock_1Hz" )
      wire#w2
      Coil( #drivesOn )
   END_RUNG
   RUNG wire#w1
      Contact( #periReady )
   END_RUNG wire#w2
   RUNG wire#w1
      Coil( #moveEnable )
   END_RUNG
   RUNG wire#w1
      Move(in := #JobNrReq, out1 => #jobNr)
   END_RUNG
   RUNG wire#powerrail
      Coil( #moveEnable )
   END_RUNG
   // the same network as SCL:
   #drivesOn := #StartAllowed AND ((NOT #periReady AND "Clock_1Hz") OR #periReady);
   #moveEnable := #StartAllowed;
   IF #StartAllowed THEN #jobNr := #JobNrReq; END_IF;
   #moveEnable := TRUE;
END_REGION

REGION Network 3: Reset alarm
   RUNG wire#powerrail
      Contact( #StartAllowed )
      Contact( #periReady )
      Contact( #stopMess )
      Contact( "Clock_1Hz" )
      Coil( #confMess )
   END_RUNG
   // the same network as SCL:
   #confMess := #StartAllowed AND #periReady AND #stopMess AND "Clock_1Hz";
END_REGION

REGION Network 4: Start signal
   RUNG wire#powerrail
      Contact( #StartAllowed )
      I_Contact( #stopMess )
      I_Contact( #progAct )
      Contact( #moveEnable )
      Contact( #periReady )
      Contact( "Clock_1Hz" )
      Coil( #ExtStart )
   END_RUNG
   // the same network as SCL:
   #ExtStart := #StartAllowed AND NOT #stopMess AND NOT #progAct AND #moveEnable AND #periReady AND "Clock_1Hz";
END_REGION
END_FUNCTION_BLOCK

FUNCTION_BLOCK "HydraulicMain"
{ S7_Optimized_Access := 'TRUE' }
VERSION : 0.1
   VAR 
      HydraulicCylinder_LeftCupforming : "HydraulicCylinder";
      HydraulicCylinder_RightCupforming : "HydraulicCylinder";
      VH1StatusOld : "UDT_Cylinder";
      VH2StatusOld : "UDT_Cylinder";
      VH3StatusOld : "UDT_Cylinder";
      VH4StatusOld : "UDT_Cylinder";
      FittingCycle_InstanceCupformingLeft : "FittingCycle";
      FittingCycle_InstanceCupformingRight : "FittingCycle";
      R_TRIG_Instance {InstructionName := 'R_TRIG'; LibVersion := '1.0'} : R_TRIG;
      R_TRIG_Instance_1 {InstructionName := 'R_TRIG'; LibVersion := '1.0'} : R_TRIG;
      R_TRIG_Instance_2 {InstructionName := 'R_TRIG'; LibVersion := '1.0'} : R_TRIG;
      R_TRIG_Instance_3 {InstructionName := 'R_TRIG'; LibVersion := '1.0'} : R_TRIG;
      HydraulicMotor_Instance : "HydraulicMotor";
      dummyCylinderLeft { ExternalAccessible := 'False'; ExternalVisible := 'False'; ExternalWritable := 'False'; S7_SetPoint := 'False'} : "UDT_Cylinder";
      dummyCylinderRight : "UDT_Cylinder";
   END_VAR

   VAR_TEMP 
      i : Int;
   END_VAR


BEGIN
	REGION cylinders data
	    "DevicesData".cupformingLeft_cylinder.Position := "AnalogData".InputResults[3];
	    "DevicesData".cupformingRight_cylinder.Position := "AnalogData".InputResults[4];
	    "DevicesData".cupformingLeft_cylinder.Force := "DevicesData".Digiforce1.ActualForce;
	    "DevicesData".cupformingRight_cylinder.Force := "DevicesData".Digiforce2.ActualForce;
	    "DevicesData".cupformingLeft_cylinder.HAxis := "DevicesData".Digiforce1.ActualWay;
	    "DevicesData".cupformingRight_cylinder.HAxis := "DevicesData".Digiforce2.ActualWay;
	END_REGION
	
	REGION common pressure
	    "DevicesData".cupformingRight_cylinder.PressureCmd := "DevicesData".cupformingLeft_cylinder.PressureCmd;
	    "DevicesData".CupformingPressure := "DevicesData".cupformingLeft_cylinder.PressureCmd;
	END_REGION
	REGION stop cylinders IF reduction valve is off
	    IF NOT "qHydraulicReductionValveCupforming" THEN
	        "DevicesData".cupformingLeft_cylinder.Status.ToFp := TRUE;
	        "DevicesData".cupformingRight_cylinder.Status.ToFp := TRUE;
	    END_IF;
	END_REGION
	REGION dummy cylinders
	    #dummyCylinderLeft.InBp := #dummyCylinderLeft.ToBp;
	    #dummyCylinderLeft.InWp := #dummyCylinderLeft.ToWp;
	    #dummyCylinderRight.InBp := #dummyCylinderRight.ToBp;
	    #dummyCylinderRight.InWp := #dummyCylinderRight.ToWp;
	END_REGION
	
	REGION cupforming left - VH1
	    #HydraulicCylinder_LeftCupforming(HydraulicActive := "safety_signals"."3L+" AND "qHydraulicKM20"(* AND "qHydraulicMotorStart" AND "qHydraulicReduction valve"*),
	                                      BasicPositionMin := "StationParameters".VH1BasicPositionMin,
	                                      BasicPositionMax := "StationParameters".VH1BasicPositionMax,
	                                      MaxPosition := "StationParameters".VH1MaxPosition,
	                                      ManualCommand := "HMIData".ManualCommand,
	                                      CylinderNumber := 3,
	                                      data := "DevicesData".cupformingLeft_cylinder);
	    #FittingCycle_InstanceCupformingLeft(parameters := "DB_ProductionProgramActual".Program.CupformingParametersLeft,
	                                         basicPosition := "DevicesData".cupformingLeft_cylinder.Status.InBp AND
	                                         "DevicesData".Cylinders["MM302_ShiftingSupportLeft"].InBp AND
	                                         "DevicesData".Cylinders["MM352_ShiftWedgeLeft"].InBp AND
	                                         "DevicesData".Cylinders["MM3100_SidememberSupport"].InBp,
	                                         MaxPosition := "StationParameters".VH1MaxPosition,
	                                         endStopCylinderActive := true,
	                                         shiftSupportToWork := "DB_ProductionProgramActual".Program.MechanicalType = 0,
	                                         rivetSensor := TRUE,
	                                         rivetStatusOtherCylinder := 1,
	                                         HydraulicCylinder := "DevicesData".cupformingLeft_cylinder,
	                                         dataFitting := "DevicesData".cupformingLeft_cycle,
	                                         dataDigiforce := "DevicesData".Digiforce1,
	                                         stopperForWedgeCylinder := "DevicesData".Cylinders["MM306_MovingStopLeft"],
	                                         supportCylinder := "DevicesData".Cylinders["MM302_ShiftingSupportLeft"],
	                                         wedgeCylinder := "DevicesData".Cylinders["MM352_ShiftWedgeLeft"],
	                                         MeasuredData := "AutoInfo".PartMeasuredData.LeftCupforming);
	END_REGION
	REGION cupforming right - VH2
	    #HydraulicCylinder_RightCupforming(HydraulicActive := "safety_signals"."3L+" AND "qHydraulicKM20"(* AND "qHydraulicMotorStart" AND "qHydraulicReduction valve"*),
	                                       BasicPositionMin := "StationParameters".VH2BasicPositionMin,
	                                       BasicPositionMax := "StationParameters".VH2BasicPositionMax,
	                                       MaxPosition := "StationParameters".VH2MaxPosition,
	                                       ManualCommand := "HMIData".ManualCommand,
	                                       CylinderNumber := 4,
	                                       data := "DevicesData".cupformingRight_cylinder);
	    #FittingCycle_InstanceCupformingRight(parameters := "DB_ProductionProgramActual".Program.CupformingParametersRight,
	                                          basicPosition := "DevicesData".cupformingRight_cylinder.Status.InBp AND
	                                          "DevicesData".Cylinders["MM300_ShiftingSupportRight"].InBp AND
	                                          "DevicesData".Cylinders["MM350_ShiftWedgeRight"].InBp AND
	                                          "DevicesData".Cylinders["MM3100_SidememberSupport"].InBp,
	                                          MaxPosition := "StationParameters".VH2MaxPosition,
	                                          endStopCylinderActive := true,
	                                          shiftSupportToWork := "DB_ProductionProgramActual".Program.MechanicalType = 1,
	                                          rivetSensor := TRUE,
	                                          rivetStatusOtherCylinder := 1,
	                                          HydraulicCylinder := "DevicesData".cupformingRight_cylinder,
	                                          dataFitting := "DevicesData".cupformingRight_cycle,
	                                          dataDigiforce := "DevicesData".Digiforce2,
	                                          stopperForWedgeCylinder := "DevicesData".Cylinders["MM304_MovingStopRight"],
	                                          supportCylinder := "DevicesData".Cylinders["MM300_ShiftingSupportRight"],
	                                          wedgeCylinder := "DevicesData".Cylinders["MM350_ShiftWedgeRight"],
	                                          MeasuredData := "AutoInfo".PartMeasuredData.RightCupforming);
	END_REGION
	
	REGION cycles handshake
	    IF "SystemHMI".AutomaticMode THEN
	        IF "DevicesData".cupformingLeft_cycle.InPreposition AND "DevicesData".cupformingRight_cycle.InPreposition THEN
	            "DevicesData".cupformingLeft_cycle.ContinueFitting := TRUE;
	            "DevicesData".cupformingRight_cycle.ContinueFitting := TRUE;
	        END_IF;
	        IF "DevicesData".cupformingLeft_cycle.Returning AND "DevicesData".cupformingRight_cycle.Returning THEN
	            "DevicesData".cupformingLeft_cycle.ContinueReturn := TRUE;
	            "DevicesData".cupformingRight_cycle.ContinueReturn := TRUE;
	        END_IF;
	        "DevicesData".cupformingLeft_cycle.continueWithSupportToWork := TRUE;
	        "DevicesData".cupformingRight_cycle.continueWithSupportToWork := TRUE;
	    END_IF;
	    
	    IF "SystemHMI".ManualMode THEN
	        "DevicesData".cupformingLeft_cycle.ContinueFitting := true;
	        "DevicesData".cupformingLeft_cycle.ContinueReturn := true;
	        "DevicesData".cupformingLeft_cycle.continueWithSupportToWork := true;
	        "DevicesData".cupformingRight_cycle.ContinueFitting := true;
	        "DevicesData".cupformingRight_cycle.ContinueReturn := true;
	        "DevicesData".cupformingRight_cycle.continueWithSupportToWork := true;
	    END_IF;
	END_REGION
	
	REGION manual mode
	//Start fitting in manual mode
	    IF "SystemHMI".ManualMode THEN
	        IF "HMIData".ManualCommand = 5101 THEN
	            "DevicesData".rivetingLeft_cycle.Start := true;
	        END_IF;
	        IF "HMIData".ManualCommand = 6101 THEN
	            "DevicesData".rivetingLeft_cycle.Start := false;
	        END_IF;
	        IF "HMIData".ManualCommand = 5102 THEN
	            "DevicesData".rivetingRight_cycle.Start := true;
	        END_IF;
	        IF "HMIData".ManualCommand = 6102 THEN
	            "DevicesData".rivetingRight_cycle.Start := false;
	        END_IF;
	        
	        IF "HMIData".ManualCommand = 5103 THEN
	            "DevicesData".cupformingLeft_cycle.Start := true;
	        END_IF;
	        IF "HMIData".ManualCommand = 6103 THEN
	            "DevicesData".cupformingLeft_cycle.Start := false;
	        END_IF;
	        IF "HMIData".ManualCommand = 5104 THEN
	            "DevicesData".cupformingRight_cycle.Start := true;
	        END_IF;
	        IF "HMIData".ManualCommand = 6104 THEN
	            "DevicesData".cupformingRight_cycle.Start := false;
	        END_IF;
	    END_IF;
	    
	    //Finished cycle detection in manual mode
	    #R_TRIG_Instance(CLK := "DevicesData".rivetingLeft_cycle.Done);
	    #R_TRIG_Instance_1(CLK := "DevicesData".rivetingRight_cycle.Done);
	    #R_TRIG_Instance_2(CLK := "DevicesData".cupformingLeft_cycle.Done);
	    #R_TRIG_Instance_3(CLK := "DevicesData".cupformingRight_cycle.Done);
	    
	    //Copy part errors after finishing cycle
	    
	    IF #R_TRIG_Instance.Q THEN
	        FOR #i := 1 TO 8 DO
	            "Alarms".PartErrorsHMI[#i + 9] := "DevicesData".rivetingLeft_cycle.PartErrors[#i];
	        END_FOR;
	    END_IF;
	    IF #R_TRIG_Instance_1.Q THEN
	        FOR #i := 1 TO 8 DO
	            "Alarms".PartErrorsHMI[#i + 19] := "DevicesData".rivetingRight_cycle.PartErrors[#i];
	        END_FOR;
	    END_IF;
	    IF #R_TRIG_Instance_2.Q THEN
	        FOR #i := 1 TO 8 DO
	            "Alarms".PartErrorsHMI[#i + 29] := "DevicesData".cupformingLeft_cycle.PartErrors[#i];
	        END_FOR;
	    END_IF;
	    IF #R_TRIG_Instance_3.Q THEN
	        FOR #i := 1 TO 8 DO
	            "Alarms".PartErrorsHMI[#i + 39] := "DevicesData".cupformingRight_cycle.PartErrors[#i];
	        END_FOR;
	    END_IF;
	    
	    //reset cycles when mode change
	    IF "SystemHMI".ModeChanged AND
	        NOT ("ModeSelection_DB".PrevMode = "mode_3_automat" AND "ModeSelection_DB".mode.activeMode = "mode_3_automat") AND
	        NOT ("ModeSelection_DB".PrevMode = "mode_4_semiautomat" AND "ModeSelection_DB".mode.activeMode = "mode_4_semiautomat")
	    THEN
	        "DevicesData".cupformingLeft_cycle.Start := false;
	        "DevicesData".cupformingRight_cycle.Start := false;
	        "DevicesData".rivetingLeft_cycle.Start := false;
	        "DevicesData".rivetingRight_cycle.Start := false;
	    END_IF;
	END_REGION
	
	REGION hydraulic pump
	    #HydraulicMotor_Instance(cycleActiveCupforming :=
	                             #FittingCycle_InstanceCupformingLeft.cnt >= 40 AND #FittingCycle_InstanceCupformingLeft.cnt <= 105 OR
	                             #FittingCycle_InstanceCupformingRight.cnt >= 40 AND #FittingCycle_InstanceCupformingRight.cnt <= 105 OR
	                             ("sq_fitting_station_st3"."Hydraulic cylinders back".X OR "sq_fitting_station_st3"."Hydraulic cylinders back.".X) AND
	                             (NOT "DevicesData".cupformingLeft_cylinder.Status.InBp OR NOT "DevicesData".cupformingRight_cylinder.Status.InBp),
	                             cycleActiveRiveting := FALSE,
	                             temp1nok := "iOilTemperature50",
	                             temp2nok := "iOilTemperature65" OR NOT "iOilLowLevelOK" OR NOT "iOilHighLevekOK",
	                             data := "DevicesData".Hydraulic,
	                             qKM20 := "DevicesData".Hydraulic.StartMotor,
	//                             qMotor := "qHydraulicMotorStart",
	                             qValveCupforming := "qHydraulicReductionValveCupforming");
	    IF "ModeSelection_DB".mode.modeChanged THEN
	        IF "ModeSelection_DB".mode.activeMode = "mode_0_not_selected" OR
	            "ModeSelection_DB".mode.activeMode = "mode_1_manual" THEN
	            "DevicesData".Hydraulic.AutoMode := FALSE;
	        END_IF;
	    END_IF;
	    IF "sq_fitting_station_st3"."Hydraulic cylinders back".X OR
	        "sq_fitting_station_st3"."Hydraulic cylinders back.".X THEN
	        "DevicesData".cupformingLeft_cylinder.PressureCmd := "DB_ProductionProgramActual".Program.CupformingParametersLeft.ApproachForce;
	        "DevicesData".cupformingRight_cylinder.PressureCmd := "DB_ProductionProgramActual".Program.CupformingParametersRight.ApproachForce;
	        "DevicesData".cupformingLeft_cylinder.FlowCmd := "DB_ProductionProgramActual".Program.CupformingParametersLeft.ApproachSpeed;
	        "DevicesData".cupformingRight_cylinder.FlowCmd := "DB_ProductionProgramActual".Program.CupformingParametersRight.ApproachSpeed;
	    END_IF;
	END_REGION
	
	REGION Riveting cylinders reduction valve Manual control
	    IF "DB_MainData".HMI.ActualScreenNumber <> 11 OR NOT "SystemHMI".ManualMode THEN
	        "HydraulicManualMode".CupformingCylinderActiveHMI := false;
	    END_IF;
	    
	    IF "SystemHMI".ManualMode THEN
	        IF NOT "DevicesData".cupformingLeft_cycle.Running AND NOT "DevicesData".cupformingRight_cycle.Running THEN
	            "qHydraulicReductionValveCupforming" := "HydraulicManualMode".CupformingCylinderActiveHMI AND NOT "iOilTemperature50";
	        ELSE
	            "HydraulicManualMode".CupformingCylinderActiveHMI := false;
	        END_IF;
	    END_IF;
	    
	END_REGION
	
	REGION history
	    "FittingHistoryLeftCupforming_DB"(iNewCycle := "DevicesData".cupformingLeft_cycle.Done,
	                                      iData := "AutoInfo".PartMeasuredData.LeftCupforming);
	    "FittingHistoryRightCupforming_DB"(iNewCycle := "DevicesData".cupformingRight_cycle.Done,
	                                       iData := "AutoInfo".PartMeasuredData.RightCupforming);
	END_REGION
	
	
END_FUNCTION_BLOCK

FUNCTION_BLOCK "HydraulicCylinder"   // FB17, LAD
{ S7_Optimized_Access := 'TRUE' }
VERSION : 0.1
// stored: AutoNumber true, IsIECCheckEnabled false, IsRetainMemResEnabled false, MemoryReserve 100, SetENOAutomatically false, UDAEnableTagReadback false
   VAR_INPUT
      HydraulicActive : Bool;
      BasicPositionMin : Real;
      BasicPositionMax : Real;
      MaxPosition : Real;
      ManualCommand : Int;
      CylinderNumber : Int;
   END_VAR
   VAR_IN_OUT
      data : "UDT_HydraulicCylinderData";
   END_VAR
   VAR
      dataOld : "UDT_HydraulicCylinderData";
      noCollision { S7_SetPoint := 'True'} : Bool;
      IEC_Timer_0_Instance { S7_SetPoint := 'True'} : TON_TIME;
      R_TRIG_Instance { S7_SetPoint := 'True'} : R_TRIG;
      difference { S7_SetPoint := 'True'} : Real;
      re : Real;
      IEC_Timer_0_Instance_1 { S7_SetPoint := 'True'} : TON_TIME;
      RampFunction_Instance { S7_SetPoint := 'True'} : RampFunction;
      BasicPositionMin_1mm_margin : Real;
      BasicPositionMax_1mm_margin : Real;
   END_VAR
   VAR_TEMP
      command : Int;
   END_VAR
   VAR_TEMP   // added for the SCL form of the ladder/FBD networks
      _w1 : Bool;
   END_VAR
BEGIN

REGION Network 1
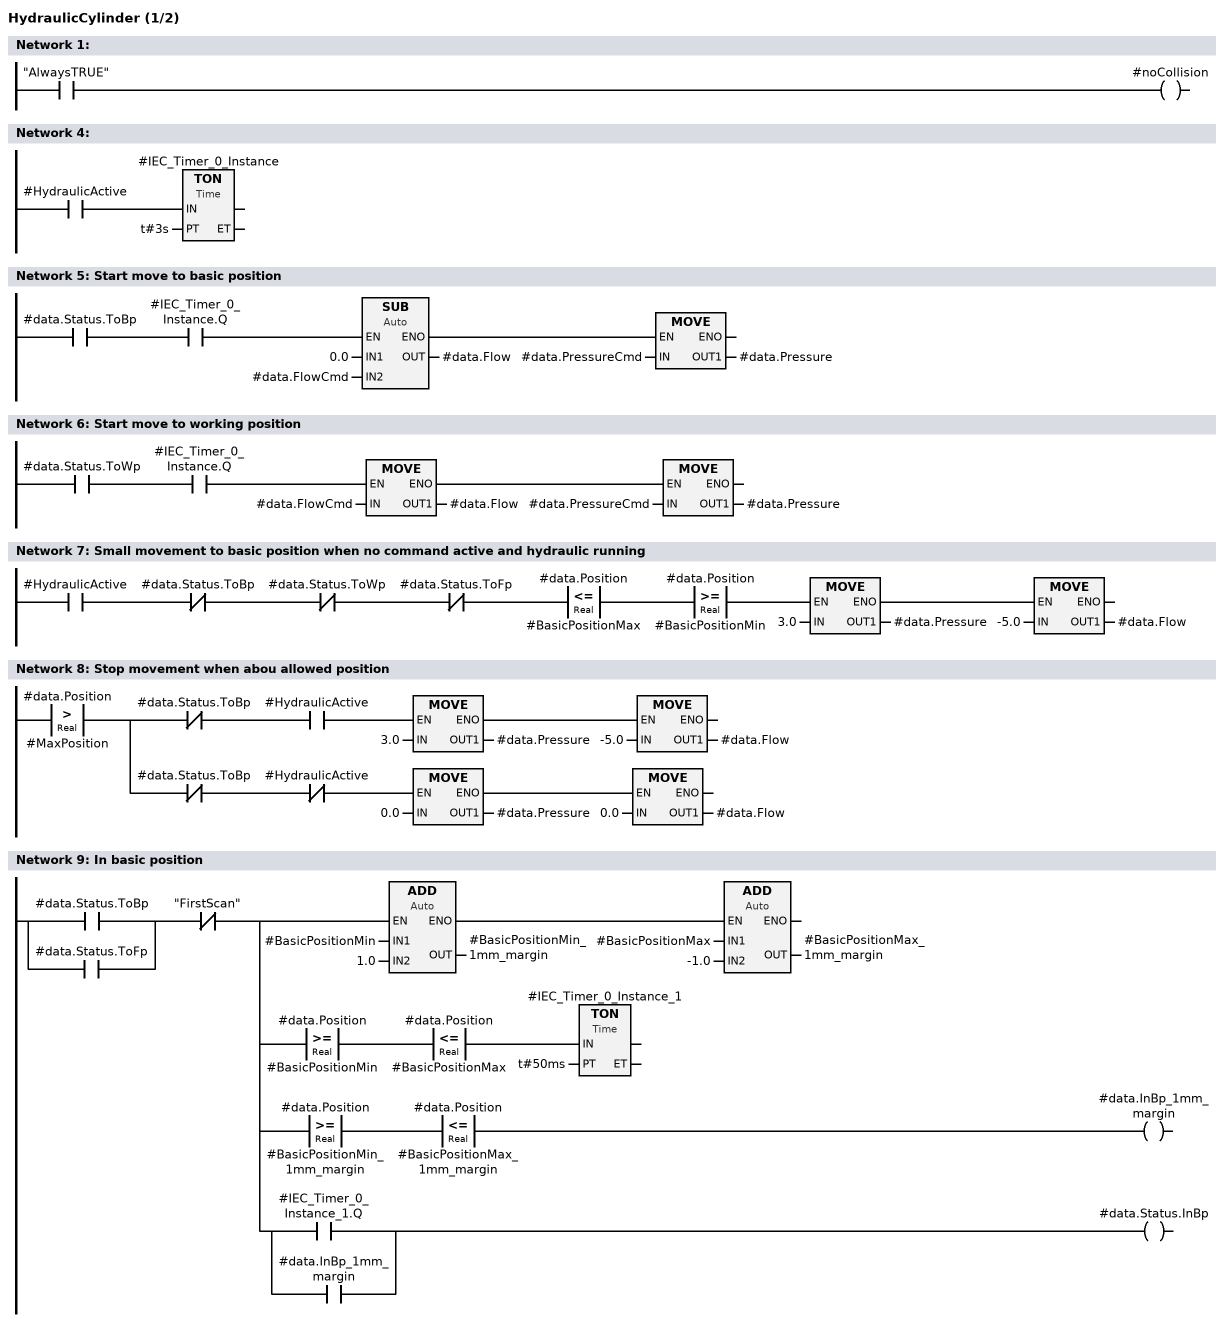
   RUNG wire#powerrail
      Contact( "AlwaysTRUE" )
      Coil( #noCollision )
   END_RUNG
   // the same network as SCL:
   #noCollision := "AlwaysTRUE";
END_REGION

REGION Network 2 (SCL)
   #command := #ManualCommand - #CylinderNumber;

